LIN {X 0,Y 226.727,Z 813.985,A -85,B 0,C 180,E1 10943.796,E2 10943.796} C_VEL
LIN {X 0,Y 213.913,Z 842.664,A -85,B 0,C 180,E1 10939.312,E2 10939.312} C_VEL
LIN {X 0,Y 200.082,Z 866.438,A -85,B 0,C 180,E1 10933.575,E2 10933.575} C_VEL
LIN {X 0,Y 185.889,Z 886.486,A -85,B 0,C 180,E1 10925.902,E2 10925.902} C_VEL
LIN {X 0,Y 173.334,Z 901.965,A -85,B 0,C 180,E1 10915.797,E2 10915.797} C_VEL
LIN {X 0,Y 166.126,Z 910.389,A -85,B 0,C 180,E1 10905.806,E2 10905.806} C_VEL
LIN {X 0,Y 162.746,Z 914.405,A -85,B 0,C 180,E1 10895.312,E2 10895.312} C_VEL
LIN {X 0,Y 162.741,Z 914.431,A -85,B 0,C 180,E1 10884.671,E2 10884.671} C_VEL
LIN {X 0,Y 167.118,Z 909.261,A -85,B 0,C 180,E1 10872.286,E2 10872.286} C_VEL
LIN {X 0,Y 175.74,Z 899.256,A -85,B 0,C 180,E1 10861.809,E2 10861.809} C_VEL
LIN {X 0,Y 188.32,Z 883.429,A -85,B 0,C 180,E1 10852.545,E2 10852.545} C_VEL
LIN {X 0,Y 202.037,Z 863.615,A -85,B 0,C 180,E1 10845.474,E2 10845.474} C_VEL
LIN {X 0,Y 213.679,Z 843.483,A -85,B 0,C 180,E1 10840.733,E2 10840.733} C_VEL
LIN {X 0,Y 213.822,Z 841.755,A -85,B 0,C 180,E1 10840.089,E2 10840.089} C_VEL
LIN {X 0,Y 191.201,Z 854.023,A -85,B 0,C 180,E1 10834.887,E2 10834.887} C_VEL
LIN {X 0,Y 172.015,Z 863.269,A -85,B 0,C 180,E1 10827.408,E2 10827.408} C_VEL
LIN {X 0,Y 171.055,Z 864.24,A -85,B 0,C 180,E1 10826.511,E2 10826.511} C_VEL
LIN {X 0,Y 165.391,Z 887.788,A -85,B 0,C 180,E1 10817.921,E2 10817.921} C_VEL
LIN {X 0,Y 162.551,Z 906.246,A -85,B 0,C 180,E1 10807.992,E2 10807.992} C_VEL
LIN {X 0,Y 163.37,Z 919.553,A -85,B 0,C 180,E1 10797.341,E2 10797.341} C_VEL
LIN {X 0,Y 168.358,Z 927.831,A -85,B 0,C 180,E1 10787.041,E2 10787.041} C_VEL
LIN {X 0,Y 181.245,Z 932.296,A -85,B 0,C 180,E1 10775.39,E2 10775.39} C_VEL
LIN {X 0,Y 203.927,Z 931.055,A -85,B 0,C 180,E1 10764.501,E2 10764.501} C_VEL
LIN {X 0,Y 173.284,Z 950.433,A -85,B 0,C 180,E1 10749.162,E2 10749.162} C_VEL
LIN {X 0,Y 161.166,Z 962.439,A -85,B 0,C 180,E1 10732.005,E2 10732.005} C_VEL
LIN {X 0,Y 159.958,Z 966.188,A -85,B 0,C 180,E1 10720.884,E2 10720.884} C_VEL
LIN {X 0,Y 161.306,Z 966.713,A -85,B 0,C 180,E1 10710.008,E2 10710.008} C_VEL
LIN {X 0,Y 160.431,Z 963.91,A -85,B 0,C 180,E1 10699.165,E2 10699.165} C_VEL
LIN {X 0,Y 161.685,Z 956.022,A -85,B 0,C 180,E1 10688.087,E2 10688.087} C_VEL
LIN {X 0,Y 167.216,Z 942.935,A -85,B 0,C 180,E1 10677.225,E2 10677.225} C_VEL
LIN {X 0,Y 177.544,Z 923.702,A -85,B 0,C 180,E1 10667.168,E2 10667.168} C_VEL
LIN {X 0,Y 187.92,Z 904.945,A -85,B 0,C 180,E1 10660.657,E2 10660.657} C_VEL
LIN {X 0,Y 191.12,Z 893.404,A -85,B 0,C 180,E1 10656.782,E2 10656.782} C_VEL
LIN {X 0,Y 194.609,Z 881.1,A -85,B 0,C 180,E1 10653.221,E2 10653.221} C_VEL
LIN {X 0,Y 208.193,Z 850.796,A -85,B 0,C 180,E1 10648.474,E2 10648.474} C_VEL
LIN {X 0,Y 214.588,Z 832.369,A -85,B 0,C 180,E1 10646.423,E2 10646.423} C_VEL
LIN {X 0,Y 212.245,Z 794.393,A -85,B 0,C 180,E1 10636.132,E2 10636.132} C_VEL
LIN {X 0,Y 211.18,Z 759.787,A -85,B 0,C 180,E1 10626.677,E2 10626.677} C_VEL
LIN {X 0,Y 209.986,Z 755.134,A -85,B 0,C 180,E1 10621.038,E2 10621.038} C_VEL
LIN {X 0,Y 210.012,Z 756.128,A -85,B 0,C 180,E1 10615.631,E2 10615.631} C_VEL
LIN {X 0,Y 212.29,Z 763.26,A -85,B 0,C 180,E1 10607.698,E2 10607.698} C_VEL
LIN {X 0,Y 216.099,Z 774.144,A -85,B 0,C 180,E1 10600.64,E2 10600.64} C_VEL
LIN {X 0,Y 220.106,Z 790.379,A -85,B 0,C 180,E1 10593.547,E2 10593.547} C_VEL
LIN {X 0,Y 221.781,Z 807.929,A -85,B 0,C 180,E1 10587.791,E2 10587.791} C_VEL
LIN {X 0,Y 221.074,Z 818.297,A -85,B 0,C 180,E1 10584.988,E2 10584.988} C_VEL
LIN {X 0,Y 207.742,Z 846.1,A -85,B 0,C 180,E1 10580.508,E2 10580.508} C_VEL
LIN {X 0,Y 193.315,Z 869.391,A -85,B 0,C 180,E1 10574.624,E2 10574.624} C_VEL
LIN {X 0,Y 178.912,Z 888.584,A -85,B 0,C 180,E1 10566.924,E2 10566.924} C_VEL
LIN {X 0,Y 166.33,Z 903.215,A -85,B 0,C 180,E1 10556.969,E2 10556.969} C_VEL
LIN {X 0,Y 158.629,Z 911.638,A -85,B 0,C 180,E1 10546.574,E2 10546.574} C_VEL
LIN {X 0,Y 154.985,Z 915.652,A -85,B 0,C 180,E1 10535.579,E2 10535.579} C_VEL
LIN {X 0,Y 154.979,Z 915.678,A -85,B 0,C 180,E1 10524.404,E2 10524.404} C_VEL
LIN {X 0,Y 158.624,Z 911.712,A -85,B 0,C 180,E1 10513.408,E2 10513.408} C_VEL
LIN {X 0,Y 167.577,Z 901.928,A -85,B 0,C 180,E1 10501.776,E2 10501.776} C_VEL
LIN {X 0,Y 180.674,Z 886.595,A -85,B 0,C 180,E1 10491.966,E2 10491.966} C_VEL
LIN {X 0,Y 195.534,Z 866.419,A -85,B 0,C 180,E1 10484.319,E2 10484.319} C_VEL
LIN {X 0,Y 204.326,Z 852.412,A -85,B 0,C 180,E1 10480.722,E2 10480.722} C_VEL
LIN {X 0,Y 203.321,Z 851.933,A -85,B 0,C 180,E1 10480.046,E2 10480.046} C_VEL
LIN {X 0,Y 175.969,Z 865.016,A -85,B 0,C 180,E1 10472.393,E2 10472.393} C_VEL
LIN {X 0,Y 161.557,Z 871.91,A -85,B 0,C 180,E1 10464.839,E2 10464.839} C_VEL
LIN {X 0,Y 156.121,Z 895.313,A -85,B 0,C 180,E1 10454.816,E2 10454.816} C_VEL
LIN {X 0,Y 154.496,Z 912.023,A -85,B 0,C 180,E1 10444.188,E2 10444.188} C_VEL
LIN {X 0,Y 157.443,Z 925.022,A -85,B 0,C 180,E1 10431.723,E2 10431.723} C_VEL
LIN {X 0,Y 167.963,Z 932.703,A -85,B 0,C 180,E1 10418.928,E2 10418.928} C_VEL
LIN {X 0,Y 181.887,Z 934.6,A -85,B 0,C 180,E1 10410.137,E2 10410.137} C_VEL
LIN {X 0,Y 193.717,Z 934.19,A -85,B 0,C 180,E1 10404.961,E2 10404.961} C_VEL
LIN {X 0,Y 180.096,Z 941.694,A -85,B 0,C 180,E1 10398.961,E2 10398.961} C_VEL
LIN {X 0,Y 156.809,Z 957.546,A -85,B 0,C 180,E1 10379.977,E2 10379.977} C_VEL
LIN {X 0,Y 152.404,Z 963.144,A -85,B 0,C 180,E1 10367.29,E2 10367.29} C_VEL
LIN {X 0,Y 152.716,Z 964.845,A -85,B 0,C 180,E1 10355.68,E2 10355.68} C_VEL
LIN {X 0,Y 153.484,Z 965.461,A -85,B 0,C 180,E1 10350.009,E2 10350.009} C_VEL
LIN {X 0,Y 152.596,Z 963.789,A -85,B 0,C 180,E1 10341.501,E2 10341.501} C_VEL
LIN {X 0,Y 153.161,Z 957.796,A -85,B 0,C 180,E1 10330.686,E2 10330.686} C_VEL
LIN {X 0,Y 158.676,Z 944.628,A -85,B 0,C 180,E1 10317.784,E2 10317.784} C_VEL
LIN {X 0,Y 169.876,Z 925.215,A -85,B 0,C 180,E1 10306.502,E2 10306.502} C_VEL
LIN {X 0,Y 183.892,Z 901.354,A -85,B 0,C 180,E1 10298.019,E2 10298.019} C_VEL
LIN {X 0,Y 194.609,Z 881.1,A -85,B 0,C 180,E1 10293.221,E2 10293.221} C_VEL
LIN {X 0,Y 198.343,Z 868.128,A -85,B 0,C 180,E1 10289.936,E2 10289.936} C_VEL
LIN {X 0,Y 201.523,Z 856.291,A -85,B 0,C 180,E1 10287.312,E2 10287.312} C_VEL
LIN {X 0,Y 202.307,Z 854.439,A -85,B 0,C 180,E1 10287.059,E2 10287.059} C_VEL
LIN {X 0,Y 209.588,Z 835.114,A -85,B 0,C 180,E1 10284.745,E2 10284.745} C_VEL
LIN {X 0,Y 209.065,Z 796.132,A -85,B 0,C 180,E1 10273.869,E2 10273.869} C_VEL
LIN {X 0,Y 209.527,Z 766.811,A -85,B 0,C 180,E1 10265.433,E2 10265.433} C_VEL
LIN {X 0,Y 208.848,Z 762.923,A -85,B 0,C 180,E1 10261.044,E2 10261.044} C_VEL
LIN {X 0,Y 208.74,Z 763.849,A -85,B 0,C 180,E1 10255.994,E2 10255.994} C_VEL
LIN {X 0,Y 210.355,Z 770.807,A -85,B 0,C 180,E1 10248.108,E2 10248.108} C_VEL
LIN {X 0,Y 213.703,Z 782.943,A -85,B 0,C 180,E1 10240.319,E2 10240.319} C_VEL
LIN {X 0,Y 216.52,Z 799.927,A -85,B 0,C 180,E1 10233.076,E2 10233.076} C_VEL
LIN {X 0,Y 216.689,Z 817.671,A -85,B 0,C 180,E1 10227.318,E2 10227.318} C_VEL
LIN {X 0,Y 215.236,Z 822.861,A -85,B 0,C 180,E1 10226.235,E2 10226.235} C_VEL
LIN {X 0,Y 201.672,Z 849.417,A -85,B 0,C 180,E1 10221.775,E2 10221.775} C_VEL
LIN {X 0,Y 185.68,Z 873.66,A -85,B 0,C 180,E1 10215.318,E2 10215.318} C_VEL
LIN {X 0,Y 169.985,Z 892.966,A -85,B 0,C 180,E1 10206.746,E2 10206.746} C_VEL
LIN {X 0,Y 158.14,Z 905.758,A -85,B 0,C 180,E1 10196.945,E2 10196.945} C_VEL
LIN {X 0,Y 149.8,Z 914.308,A -85,B 0,C 180,E1 10184.578,E2 10184.578} C_VEL
LIN {X 0,Y 146.893,Z 917.424,A -85,B 0,C 180,E1 10169.991,E2 10169.991} C_VEL
LIN {X 0,Y 149.79,Z 914.373,A -85,B 0,C 180,E1 10155.403,E2 10155.403} C_VEL
LIN {X 0,Y 158.099,Z 905.884,A -85,B 0,C 180,E1 10143.029,E2 10143.029} C_VEL
LIN {X 0,Y 170.757,Z 892.19,A -85,B 0,C 180,E1 10132.662,E2 10132.662} C_VEL
LIN {X 0,Y 185.618,Z 873.941,A -85,B 0,C 180,E1 10124.643,E2 10124.643} C_VEL
LIN {X 0,Y 194.654,Z 861.037,A -85,B 0,C 180,E1 10120.801,E2 10120.801} C_VEL
LIN {X 0,Y 194.758,Z 860.103,A -85,B 0,C 180,E1 10120.335,E2 10120.335} C_VEL
LIN {X 0,Y 166.102,Z 872.724,A -85,B 0,C 180,E1 10111.475,E2 10111.475} C_VEL
LIN {X 0,Y 152.112,Z 878.872,A -85,B 0,C 180,E1 10102.977,E2 10102.977} C_VEL
LIN {X 0,Y 147.54,Z 900.094,A -85,B 0,C 180,E1 10092.559,E2 10092.559} C_VEL
LIN {X 0,Y 146.839,Z 915.669,A -85,B 0,C 180,E1 10081.459,E2 10081.459} C_VEL
LIN {X 0,Y 151.324,Z 927.878,A -85,B 0,C 180,E1 10068.484,E2 10068.484} C_VEL
LIN {X 0,Y 160.744,Z 934.107,A -85,B 0,C 180,E1 10057.934,E2 10057.934} C_VEL
LIN {X 0,Y 175.327,Z 936.65,A -85,B 0,C 180,E1 10048.899,E2 10048.899} C_VEL
LIN {X 0,Y 184.424,Z 936.772,A -85,B 0,C 180,E1 10044.924,E2 10044.924} C_VEL
LIN {X 0,Y 153.363,Z 953.588,A -85,B 0,C 180,E1 10026.196,E2 10026.196} C_VEL
LIN {X 0,Y 144.74,Z 961.456,A -85,B 0,C 180,E1 10008.237,E2 10008.237} C_VEL
LIN {X 0,Y 144.879,Z 963.376,A -85,B 0,C 180,E1 9995.988,E2 9995.988} C_VEL
LIN {X 0,Y 145.641,Z 964.206,A -85,B 0,C 180,E1 9990.009,E2 9990.009} C_VEL
LIN {X 0,Y 144.741,Z 962.518,A -85,B 0,C 180,E1 9981.036,E2 9981.036} C_VEL
LIN {X 0,Y 145.65,Z 955.918,A -85,B 0,C 180,E1 9968.842,E2 9968.842} C_VEL
LIN {X 0,Y 151.824,Z 943.101,A -85,B 0,C 180,E1 9955.962,E2 9955.962} C_VEL
LIN {X 0,Y 163.881,Z 923.872,A -85,B 0,C 180,E1 9944.479,E2 9944.479} C_VEL
LIN {X 0,Y 179.118,Z 899.607,A -85,B 0,C 180,E1 9935.789,E2 9935.789} C_VEL
LIN {X 0,Y 194.276,Z 871.816,A -85,B 0,C 180,E1 9929.669,E2 9929.669} C_VEL
LIN {X 0,Y 202.307,Z 854.439,A -85,B 0,C 180,E1 9927.059,E2 9927.059} C_VEL
LIN {X 0,Y 205,Z 843.954,A -85,B 0,C 180,E1 9924.987,E2 9924.987} C_VEL
LIN {X 0,Y 204.883,Z 828.509,A -85,B 0,C 180,E1 9920.286,E2 9920.286} C_VEL
LIN {X 0,Y 206.718,Z 788.673,A -85,B 0,C 180,E1 9908.8,E2 9908.8} C_VEL
LIN {X 0,Y 207.774,Z 773.916,A -85,B 0,C 180,E1 9904.435,E2 9904.435} C_VEL
LIN {X 0,Y 207.328,Z 770.591,A -85,B 0,C 180,E1 9900.009,E2 9900.009} C_VEL
LIN {X 0,Y 207.147,Z 771.755,A -85,B 0,C 180,E1 9896.094,E2 9896.094} C_VEL
LIN {X 0,Y 208.271,Z 778.584,A -85,B 0,C 180,E1 9888.253,E2 9888.253} C_VEL
LIN {X 0,Y 210.52,Z 789.744,A -85,B 0,C 180,E1 9881.001,E2 9881.001} C_VEL
LIN {X 0,Y 212.335,Z 806.553,A -85,B 0,C 180,E1 9873.642,E2 9873.642} C_VEL
LIN {X 0,Y 211.603,Z 822.257,A -85,B 0,C 180,E1 9868.367,E2 9868.367} C_VEL
LIN {X 0,Y 197.579,Z 849.652,A -85,B 0,C 180,E1 9863.768,E2 9863.768} C_VEL
LIN {X 0,Y 181.409,Z 873.398,A -85,B 0,C 180,E1 9857.574,E2 9857.574} C_VEL
LIN {X 0,Y 165.74,Z 892.092,A -85,B 0,C 180,E1 9849.585,E2 9849.585} C_VEL
LIN {X 0,Y 152.575,Z 905.713,A -85,B 0,C 180,E1 9839.629,E2 9839.629} C_VEL
LIN {X 0,Y 143.735,Z 914.135,A -85,B 0,C 180,E1 9828.349,E2 9828.349} C_VEL
LIN {X 0,Y 139.494,Z 918.143,A -85,B 0,C 180,E1 9816.201,E2 9816.201} C_VEL
LIN {X 0,Y 139.489,Z 918.168,A -85,B 0,C 180,E1 9803.78,E2 9803.78} C_VEL
LIN {X 0,Y 144.98,Z 913,A -85,B 0,C 180,E1 9789.461,E2 9789.461} C_VEL
LIN {X 0,Y 155.452,Z 903,A -85,B 0,C 180,E1 9777.719,E2 9777.719} C_VEL
LIN {X 0,Y 170.602,Z 886.824,A -85,B 0,C 180,E1 9767.576,E2 9767.576} C_VEL
LIN {X 0,Y 185.665,Z 867.852,A -85,B 0,C 180,E1 9760.539,E2 9760.539} C_VEL
LIN {X 0,Y 158.547,Z 878.967,A -85,B 0,C 180,E1 9751.551,E2 9751.551} C_VEL
LIN {X 0,Y 142.622,Z 886.104,A -85,B 0,C 180,E1 9740.5,E2 9740.5} C_VEL
LIN {X 0,Y 138.954,Z 906.759,A -85,B 0,C 180,E1 9728.573,E2 9728.573} C_VEL
LIN {X 0,Y 140.15,Z 922.158,A -85,B 0,C 180,E1 9715.355,E2 9715.355} C_VEL
LIN {X 0,Y 147.832,Z 932.466,A -85,B 0,C 180,E1 9702.156,E2 9702.156} C_VEL
LIN {X 0,Y 160.559,Z 937.417,A -85,B 0,C 180,E1 9691.96,E2 9691.96} C_VEL
LIN {X 0,Y 173.678,Z 938.921,A -85,B 0,C 180,E1 9685.426,E2 9685.426} C_VEL
LIN {X 0,Y 169.786,Z 940.993,A -85,B 0,C 180,E1 9683.136,E2 9683.136} C_VEL
LIN {X 0,Y 142.018,Z 955.389,A -85,B 0,C 180,E1 9662.104,E2 9662.104} C_VEL
LIN {X 0,Y 137.107,Z 959.712,A -85,B 0,C 180,E1 9649.291,E2 9649.291} C_VEL
LIN {X 0,Y 137.004,Z 962.11,A -85,B 0,C 180,E1 9636.334,E2 9636.334} C_VEL
LIN {X 0,Y 137.817,Z 962.955,A -85,B 0,C 180,E1 9630.01,E2 9630.01} C_VEL
LIN {X 0,Y 136.997,Z 961.861,A -85,B 0,C 180,E1 9622.521,E2 9622.521} C_VEL
LIN {X 0,Y 137.676,Z 955.704,A -85,B 0,C 180,E1 9609.191,E2 9609.191} C_VEL
LIN {X 0,Y 144.382,Z 942.776,A -85,B 0,C 180,E1 9594.921,E2 9594.921} C_VEL
LIN {X 0,Y 156.779,Z 924.445,A -85,B 0,C 180,E1 9583.255,E2 9583.255} C_VEL
LIN {X 0,Y 172.897,Z 900.6,A -85,B 0,C 180,E1 9574.244,E2 9574.244} C_VEL
LIN {X 0,Y 188.983,Z 873.115,A -85,B 0,C 180,E1 9567.963,E2 9567.963} C_VEL
LIN {X 0,Y 203.009,Z 843.146,A -85,B 0,C 180,E1 9563.79,E2 9563.79} C_VEL
LIN {X 0,Y 204.671,Z 838.218,A -85,B 0,C 180,E1 9563.142,E2 9563.142} C_VEL
LIN {X 0,Y 204.883,Z 828.509,A -85,B 0,C 180,E1 9560.286,E2 9560.286} C_VEL
LIN {X 0,Y 203.076,Z 823.273,A -85,B 0,C 180,E1 9557.349,E2 9557.349} C_VEL
LIN {X 0,Y 201.613,Z 818.034,A -85,B 0,C 180,E1 9554.362,E2 9554.362} C_VEL
LIN {X 0,Y 205.866,Z 781.149,A -85,B 0,C 180,E1 9543.686,E2 9543.686} C_VEL
LIN {X 0,Y 205.641,Z 778.298,A -85,B 0,C 180,E1 9540.009,E2 9540.009} C_VEL
LIN {X 0,Y 205.253,Z 779.601,A -85,B 0,C 180,E1 9536.189,E2 9536.189} C_VEL
LIN {X 0,Y 205.742,Z 785.492,A -85,B 0,C 180,E1 9529.094,E2 9529.094} C_VEL
LIN {X 0,Y 207.157,Z 796.128,A -85,B 0,C 180,E1 9521.869,E2 9521.869} C_VEL
LIN {X 0,Y 207.953,Z 811.662,A -85,B 0,C 180,E1 9514.779,E2 9514.779} C_VEL
LIN {X 0,Y 206.328,Z 826.737,A -85,B 0,C 180,E1 9509.637,E2 9509.637} C_VEL
LIN {X 0,Y 191.129,Z 853.898,A -85,B 0,C 180,E1 9504.99,E2 9504.99} C_VEL
LIN {X 0,Y 173.904,Z 877.537,A -85,B 0,C 180,E1 9498.445,E2 9498.445} C_VEL
LIN {X 0,Y 157.549,Z 895.682,A -85,B 0,C 180,E1 9490.008,E2 9490.008} C_VEL
LIN {X 0,Y 143.007,Z 909.498,A -85,B 0,C 180,E1 9478.34,E2 9478.34} C_VEL
LIN {X 0,Y 134.747,Z 916.806,A -85,B 0,C 180,E1 9466.249,E2 9466.249} C_VEL
LIN {X 0,Y 131.314,Z 919.916,A -85,B 0,C 180,E1 9449.99,E2 9449.99} C_VEL
LIN {X 0,Y 134.738,Z 916.868,A -85,B 0,C 180,E1 9433.73,E2 9433.73} C_VEL
LIN {X 0,Y 144.352,Z 908.378,A -85,B 0,C 180,E1 9420.216,E2 9420.216} C_VEL
LIN {X 0,Y 158.38,Z 894.939,A -85,B 0,C 180,E1 9409.393,E2 9409.393} C_VEL
LIN {X 0,Y 174.517,Z 876.994,A -85,B 0,C 180,E1 9401.21,E2 9401.21} C_VEL
LIN {X 0,Y 174.771,Z 875.76,A -85,B 0,C 180,E1 9400.339,E2 9400.339} C_VEL
LIN {X 0,Y 148.7,Z 885.676,A -85,B 0,C 180,E1 9390.473,E2 9390.473} C_VEL
LIN {X 0,Y 133.291,Z 892.73,A -85,B 0,C 180,E1 9377.697,E2 9377.697} C_VEL
LIN {X 0,Y 130.838,Z 911.752,A -85,B 0,C 180,E1 9364.947,E2 9364.947} C_VEL
LIN {X 0,Y 133.419,Z 925.288,A -85,B 0,C 180,E1 9351.859,E2 9351.859} C_VEL
LIN {X 0,Y 143.266,Z 935.045,A -85,B 0,C 180,E1 9338.355,E2 9338.355} C_VEL
LIN {X 0,Y 163.74,Z 940.562,A -85,B 0,C 180,E1 9325.494,E2 9325.494} C_VEL
LIN {X 0,Y 155.519,Z 944.277,A -85,B 0,C 180,E1 9320.935,E2 9320.935} C_VEL
LIN {X 0,Y 132.848,Z 955.272,A -85,B 0,C 180,E1 9300.13,E2 9300.13} C_VEL
LIN {X 0,Y 128.818,Z 959.953,A -85,B 0,C 180,E1 9280.131,E2 9280.131} C_VEL
LIN {X 0,Y 129.967,Z 961.7,A -85,B 0,C 180,E1 9270.01,E2 9270.01} C_VEL
LIN {X 0,Y 128.969,Z 959.951,A -85,B 0,C 180,E1 9259.902,E2 9259.902} C_VEL
LIN {X 0,Y 130.657,Z 952.957,A -85,B 0,C 180,E1 9245.731,E2 9245.731} C_VEL
LIN {X 0,Y 138.937,Z 939.53,A -85,B 0,C 180,E1 9231.364,E2 9231.364} C_VEL
LIN {X 0,Y 153.53,Z 920.01,A -85,B 0,C 180,E1 9219.466,E2 9219.466} C_VEL
LIN {X 0,Y 170.317,Z 896.326,A -85,B 0,C 180,E1 9211.041,E2 9211.041} C_VEL
LIN {X 0,Y 187.31,Z 867.911,A -85,B 0,C 180,E1 9205.027,E2 9205.027} C_VEL
LIN {X 0,Y 199.905,Z 840.965,A -85,B 0,C 180,E1 9201.358,E2 9201.358} C_VEL
LIN {X 0,Y 201.613,Z 818.034,A -85,B 0,C 180,E1 9194.362,E2 9194.362} C_VEL
LIN {X 0,Y 201.258,Z 808.666,A -85,B 0,C 180,E1 9190.141,E2 9190.141} C_VEL
LIN {X 0,Y 201.608,Z 799.366,A -85,B 0,C 180,E1 9185.888,E2 9185.888} C_VEL
LIN {X 0,Y 203.655,Z 787.68,A -85,B 0,C 180,E1 9182.132,E2 9182.132} C_VEL
LIN {X 0,Y 203.685,Z 785.928,A -85,B 0,C 180,E1 9180.009,E2 9180.009} C_VEL
LIN {X 0,Y 203.092,Z 787.336,A -85,B 0,C 180,E1 9176.282,E2 9176.282} C_VEL
LIN {X 0,Y 203.156,Z 793.391,A -85,B 0,C 180,E1 9168.953,E2 9168.953} C_VEL
LIN {X 0,Y 203.75,Z 804.239,A -85,B 0,C 180,E1 9161.793,E2 9161.793} C_VEL
LIN {X 0,Y 203.384,Z 819.154,A -85,B 0,C 180,E1 9154.991,E2 9154.991} C_VEL
LIN {X 0,Y 201.549,Z 829.956,A -85,B 0,C 180,E1 9151.27,E2 9151.27} C_VEL
LIN {X 0,Y 185.409,Z 857.148,A -85,B 0,C 180,E1 9146.527,E2 9146.527} C_VEL
LIN {X 0,Y 167.613,Z 880.165,A -85,B 0,C 180,E1 9139.92,E2 9139.92} C_VEL
LIN {X 0,Y 150.167,Z 898.312,A -85,B 0,C 180,E1 9131.019,E2 9131.019} C_VEL
LIN {X 0,Y 136.188,Z 910.746,A -85,B 0,C 180,E1 9119.899,E2 9119.899} C_VEL
LIN {X 0,Y 127.271,Z 918.054,A -85,B 0,C 180,E1 9107.232,E2 9107.232} C_VEL
LIN {X 0,Y 123.528,Z 921.161,A -85,B 0,C 180,E1 9089.989,E2 9089.989} C_VEL
LIN {X 0,Y 127.265,Z 918.116,A -85,B 0,C 180,E1 9072.745,E2 9072.745} C_VEL
LIN {X 0,Y 137.633,Z 909.623,A -85,B 0,C 180,E1 9058.602,E2 9058.602} C_VEL
LIN {X 0,Y 152.542,Z 896.182,A -85,B 0,C 180,E1 9047.486,E2 9047.486} C_VEL
LIN {X 0,Y 164.59,Z 883.784,A -85,B 0,C 180,E1 9041.331,E2 9041.331} C_VEL
LIN {X 0,Y 165.061,Z 882.615,A -85,B 0,C 180,E1 9040.474,E2 9040.474} C_VEL
LIN {X 0,Y 138.948,Z 891.913,A -85,B 0,C 180,E1 9029.237,E2 9029.237} C_VEL
LIN {X 0,Y 124.109,Z 899.442,A -85,B 0,C 180,E1 9014.057,E2 9014.057} C_VEL
LIN {X 0,Y 123.34,Z 917.32,A -85,B 0,C 180,E1 8999.984,E2 8999.984} C_VEL
LIN {X 0,Y 129.304,Z 930.762,A -85,B 0,C 180,E1 8984.763,E2 8984.763} C_VEL
LIN {X 0,Y 143.04,Z 939.043,A -85,B 0,C 180,E1 8971.646,E2 8971.646} C_VEL
LIN {X 0,Y 153.376,Z 941.636,A -85,B 0,C 180,E1 8965.792,E2 8965.792} C_VEL
LIN {X 0,Y 148.843,Z 943.879,A -85,B 0,C 180,E1 8962.521,E2 8962.521} C_VEL
LIN {X 0,Y 124.384,Z 954.338,A -85,B 0,C 180,E1 8939.044,E2 8939.044} C_VEL
LIN {X 0,Y 121.138,Z 957.497,A -85,B 0,C 180,E1 8924.438,E2 8924.438} C_VEL
LIN {X 0,Y 122.131,Z 960.447,A -85,B 0,C 180,E1 8910.011,E2 8910.011} C_VEL
LIN {X 0,Y 121.11,Z 958.673,A -85,B 0,C 180,E1 8899.239,E2 8899.239} C_VEL
LIN {X 0,Y 123.056,Z 951.914,A -85,B 0,C 180,E1 8884.594,E2 8884.594} C_VEL
LIN {X 0,Y 132.554,Z 938.203,A -85,B 0,C 180,E1 8869.122,E2 8869.122} C_VEL
LIN {X 0,Y 147.676,Z 919.567,A -85,B 0,C 180,E1 8857.381,E2 8857.381} C_VEL
LIN {X 0,Y 165.695,Z 895.689,A -85,B 0,C 180,E1 8848.781,E2 8848.781} C_VEL
LIN {X 0,Y 183.693,Z 867.076,A -85,B 0,C 180,E1 8842.771,E2 8842.771} C_VEL
LIN {X 0,Y 195.194,Z 844.041,A -85,B 0,C 180,E1 8839.659,E2 8839.659} C_VEL
LIN {X 0,Y 200.338,Z 807.167,A -85,B 0,C 180,E1 8828.223,E2 8828.223} C_VEL
LIN {X 0,Y 201.608,Z 799.366,A -85,B 0,C 180,E1 8825.888,E2 8825.888} C_VEL
LIN {X 0,Y 202.052,Z 794.509,A -85,B 0,C 180,E1 8823.274,E2 8823.274} C_VEL
LIN {X 0,Y 201.233,Z 793.796,A -85,B 0,C 180,E1 8819.352,E2 8819.352} C_VEL
LIN {X 0,Y 200.356,Z 798.48,A -85,B 0,C 180,E1 8811.347,E2 8811.347} C_VEL
LIN {X 0,Y 200.104,Z 809.277,A -85,B 0,C 180,E1 8803.369,E2 8803.369} C_VEL
LIN {X 0,Y 199.057,Z 823.221,A -85,B 0,C 180,E1 8796.56,E2 8796.56} C_VEL
LIN {X 0,Y 197.26,Z 832.396,A -85,B 0,C 180,E1 8793.083,E2 8793.083} C_VEL
LIN {X 0,Y 181.233,Z 858.388,A -85,B 0,C 180,E1 8788.579,E2 8788.579} C_VEL
LIN {X 0,Y 162.691,Z 881.413,A -85,B 0,C 180,E1 8782.027,E2 8782.027} C_VEL
LIN {X 0,Y 144.067,Z 899.822,A -85,B 0,C 180,E1 8772.869,E2 8772.869} C_VEL
LIN {X 0,Y 129.464,Z 911.997,A -85,B 0,C 180,E1 8761.625,E2 8761.625} C_VEL
LIN {X 0,Y 119.571,Z 919.489,A -85,B 0,C 180,E1 8747.755,E2 8747.755} C_VEL
LIN {X 0,Y 115.726,Z 922.409,A -85,B 0,C 180,E1 8729.989,E2 8729.989} C_VEL
LIN {X 0,Y 119.541,Z 919.558,A -85,B 0,C 180,E1 8712.272,E2 8712.272} C_VEL
LIN {X 0,Y 131.038,Z 910.869,A -85,B 0,C 180,E1 8696.825,E2 8696.825} C_VEL
LIN {X 0,Y 146.61,Z 897.68,A -85,B 0,C 180,E1 8685.58,E2 8685.58} C_VEL
LIN {X 0,Y 154.906,Z 889.825,A -85,B 0,C 180,E1 8681.347,E2 8681.347} C_VEL
LIN {X 0,Y 154.829,Z 889.112,A -85,B 0,C 180,E1 8680.452,E2 8680.452} C_VEL
LIN {X 0,Y 125.503,Z 899.245,A -85,B 0,C 180,E1 8664.867,E2 8664.867} C_VEL
LIN {X 0,Y 115.446,Z 905.38,A -85,B 0,C 180,E1 8650.037,E2 8650.037} C_VEL
LIN {X 0,Y 116.576,Z 922.415,A -85,B 0,C 180,E1 8634.413,E2 8634.413} C_VEL
LIN {X 0,Y 127.178,Z 935.713,A -85,B 0,C 180,E1 8617.303,E2 8617.303} C_VEL
LIN {X 0,Y 143.081,Z 942.177,A -85,B 0,C 180,E1 8606.042,E2 8606.042} C_VEL
LIN {X 0,Y 143.405,Z 942.879,A -85,B 0,C 180,E1 8604.8,E2 8604.8} C_VEL
LIN {X 0,Y 117.363,Z 952.354,A -85,B 0,C 180,E1 8580.966,E2 8580.966} C_VEL
LIN {X 0,Y 113.767,Z 954.82,A -85,B 0,C 180,E1 8569.084,E2 8569.084} C_VEL
LIN {X 0,Y 113.325,Z 958.296,A -85,B 0,C 180,E1 8557.664,E2 8557.664} C_VEL
LIN {X 0,Y 114.281,Z 959.191,A -85,B 0,C 180,E1 8550.012,E2 8550.012} C_VEL
LIN {X 0,Y 113.253,Z 957.392,A -85,B 0,C 180,E1 8538.482,E2 8538.482} C_VEL
LIN {X 0,Y 115.697,Z 950.602,A -85,B 0,C 180,E1 8522.85,E2 8522.85} C_VEL
LIN {X 0,Y 126.4,Z 936.877,A -85,B 0,C 180,E1 8506.661,E2 8506.661} C_VEL
LIN {X 0,Y 142.747,Z 918.226,A -85,B 0,C 180,E1 8494.707,E2 8494.707} C_VEL
LIN {X 0,Y 161.872,Z 894.369,A -85,B 0,C 180,E1 8486.212,E2 8486.212} C_VEL
LIN {X 0,Y 180.202,Z 866.578,A -85,B 0,C 180,E1 8480.498,E2 8480.498} C_VEL
LIN {X 0,Y 190.439,Z 847.75,A -85,B 0,C 180,E1 8478.05,E2 8478.05} C_VEL
LIN {X 0,Y 197.428,Z 811.558,A -85,B 0,C 180,E1 8466.504,E2 8466.504} C_VEL
LIN {X 0,Y 201.359,Z 794.465,A -85,B 0,C 180,E1 8461.083,E2 8461.083} C_VEL
LIN {X 0,Y 201.233,Z 793.796,A -85,B 0,C 180,E1 8459.352,E2 8459.352} C_VEL
LIN {X 0,Y 199.709,Z 797.895,A -85,B 0,C 180,E1 8455.806,E2 8455.806} C_VEL
LIN {X 0,Y 197.127,Z 807.529,A -85,B 0,C 180,E1 8450.044,E2 8450.044} C_VEL
LIN {X 0,Y 196.106,Z 818.27,A -85,B 0,C 180,E1 8442.664,E2 8442.664} C_VEL
LIN {X 0,Y 193.981,Z 831.199,A -85,B 0,C 180,E1 8436.517,E2 8436.517} C_VEL
LIN {X 0,Y 192.654,Z 835.756,A -85,B 0,C 180,E1 8434.848,E2 8434.848} C_VEL
LIN {X 0,Y 175.855,Z 861.602,A -85,B 0,C 180,E1 8430.312,E2 8430.312} C_VEL
LIN {X 0,Y 156.714,Z 884.038,A -85,B 0,C 180,E1 8423.738,E2 8423.738} C_VEL
LIN {X 0,Y 138.442,Z 901.071,A -85,B 0,C 180,E1 8415.07,E2 8415.07} C_VEL
LIN {X 0,Y 122.885,Z 913.246,A -85,B 0,C 180,E1 8403.534,E2 8403.534} C_VEL
LIN {X 0,Y 113.424,Z 919.852,A -85,B 0,C 180,E1 8391.423,E2 8391.423} C_VEL
LIN {X 0,Y 108.523,Z 923.134,A -85,B 0,C 180,E1 8377.981,E2 8377.981} C_VEL
LIN {X 0,Y 108.518,Z 923.157,A -85,B 0,C 180,E1 8361.994,E2 8361.994} C_VEL
LIN {X 0,Y 114.52,Z 919.195,A -85,B 0,C 180,E1 8346.701,E2 8346.701} C_VEL
LIN {X 0,Y 128.174,Z 909.415,A -85,B 0,C 180,E1 8331.808,E2 8331.808} C_VEL
LIN {X 0,Y 144.96,Z 895.633,A -85,B 0,C 180,E1 8321.446,E2 8321.446} C_VEL
LIN {X 0,Y 145.289,Z 894.893,A -85,B 0,C 180,E1 8320.68,E2 8320.68} C_VEL
LIN {X 0,Y 113.001,Z 906.13,A -85,B 0,C 180,E1 8299.483,E2 8299.483} C_VEL
LIN {X 0,Y 107.175,Z 911.261,A -85,B 0,C 180,E1 8285.03,E2 8285.03} C_VEL
LIN {X 0,Y 110.845,Z 927.119,A -85,B 0,C 180,E1 8268.2,E2 8268.2} C_VEL
LIN {X 0,Y 125.379,Z 939.242,A -85,B 0,C 180,E1 8251.207,E2 8251.207} C_VEL
LIN {X 0,Y 133.894,Z 942.516,A -85,B 0,C 180,E1 8245.687,E2 8245.687} C_VEL
LIN {X 0,Y 112.345,Z 949.6,A -85,B 0,C 180,E1 8226.28,E2 8226.28} C_VEL
LIN {X 0,Y 107.335,Z 951.551,A -85,B 0,C 180,E1 8214.961,E2 8214.961} C_VEL
LIN {X 0,Y 105.465,Z 957.027,A -85,B 0,C 180,E1 8198.239,E2 8198.239} C_VEL
LIN {X 0,Y 106.407,Z 957.932,A -85,B 0,C 180,E1 8190.012,E2 8190.012} C_VEL
LIN {X 0,Y 105.415,Z 956.111,A -85,B 0,C 180,E1 8177.613,E2 8177.613} C_VEL
LIN {X 0,Y 108.453,Z 949.288,A -85,B 0,C 180,E1 8160.869,E2 8160.869} C_VEL
LIN {X 0,Y 120.37,Z 935.636,A -85,B 0,C 180,E1 8144.016,E2 8144.016} C_VEL
LIN {X 0,Y 138.518,Z 916.507,A -85,B 0,C 180,E1 8131.691,E2 8131.691} C_VEL
LIN {X 0,Y 158.386,Z 893.047,A -85,B 0,C 180,E1 8123.521,E2 8123.521} C_VEL
LIN {X 0,Y 177.22,Z 865.708,A -85,B 0,C 180,E1 8118.074,E2 8118.074} C_VEL
LIN {X 0,Y 185.696,Z 851.026,A -85,B 0,C 180,E1 8116.203,E2 8116.203} C_VEL
LIN {X 0,Y 193.941,Z 818.36,A -85,B 0,C 180,E1 8105.546,E2 8105.546} C_VEL
LIN {X 0,Y 198.804,Z 801.186,A -85,B 0,C 180,E1 8100.01,E2 8100.01} C_VEL
LIN {X 0,Y 197.302,Z 806.266,A -85,B 0,C 180,E1 8091.212,E2 8091.212} C_VEL
LIN {X 0,Y 197.127,Z 807.529,A -85,B 0,C 180,E1 8090.044,E2 8090.044} C_VEL
LIN {X 0,Y 195.626,Z 814.036,A -85,B 0,C 180,E1 8086.757,E2 8086.757} C_VEL
LIN {X 0,Y 191.386,Z 827.879,A -85,B 0,C 180,E1 8081.669,E2 8081.669} C_VEL
LIN {X 0,Y 188.29,Z 839.04,A -85,B 0,C 180,E1 8076.702,E2 8076.702} C_VEL
LIN {X 0,Y 170.633,Z 864.678,A -85,B 0,C 180,E1 8072.161,E2 8072.161} C_VEL
LIN {X 0,Y 150.675,Z 886.857,A -85,B 0,C 180,E1 8065.503,E2 8065.503} C_VEL
LIN {X 0,Y 131.002,Z 903.917,A -85,B 0,C 180,E1 8056.305,E2 8056.305} C_VEL
LIN {X 0,Y 114.719,Z 915.676,A -85,B 0,C 180,E1 8043.978,E2 8043.978} C_VEL
LIN {X 0,Y 103.3,Z 922.9,A -85,B 0,C 180,E1 8026.975,E2 8026.975} C_VEL
LIN {X 0,Y 100.137,Z 924.901,A -85,B 0,C 180,E1 8009.987,E2 8009.987} C_VEL
LIN {X 0,Y 105.006,Z 921.928,A -85,B 0,C 180,E1 7989.207,E2 7989.207} C_VEL
LIN {X 0,Y 118.259,Z 913.365,A -85,B 0,C 180,E1 7972.675,E2 7972.675} C_VEL
LIN {X 0,Y 134.901,Z 901.008,A -85,B 0,C 180,E1 7961.479,E2 7961.479} C_VEL
LIN {X 0,Y 133.859,Z 900.796,A -85,B 0,C 180,E1 7960.174,E2 7960.174} C_VEL
LIN {X 0,Y 102.524,Z 912.15,A -85,B 0,C 180,E1 7933.7,E2 7933.7} C_VEL
LIN {X 0,Y 99.762,Z 916.984,A -85,B 0,C 180,E1 7918.897,E2 7918.897} C_VEL
LIN {X 0,Y 107.995,Z 932.843,A -85,B 0,C 180,E1 7899.537,E2 7899.537} C_VEL
LIN {X 0,Y 123.924,Z 942.16,A -85,B 0,C 180,E1 7885.768,E2 7885.768} C_VEL
LIN {X 0,Y 121.797,Z 943.134,A -85,B 0,C 180,E1 7883.663,E2 7883.663} C_VEL
LIN {X 0,Y 99.991,Z 950.246,A -85,B 0,C 180,E1 7856.936,E2 7856.936} C_VEL
LIN {X 0,Y 97.581,Z 955.752,A -85,B 0,C 180,E1 7838.91,E2 7838.91} C_VEL
LIN {X 0,Y 98.56,Z 956.677,A -85,B 0,C 180,E1 7830.013,E2 7830.013} C_VEL
LIN {X 0,Y 97.568,Z 954.823,A -85,B 0,C 180,E1 7816.599,E2 7816.599} C_VEL
LIN {X 0,Y 101.337,Z 947.971,A -85,B 0,C 180,E1 7798.602,E2 7798.602} C_VEL
LIN {X 0,Y 114.407,Z 934.598,A -85,B 0,C 180,E1 7781.279,E2 7781.279} C_VEL
LIN {X 0,Y 132.605,Z 916.932,A -85,B 0,C 180,E1 7769.495,E2 7769.495} C_VEL
LIN {X 0,Y 153.732,Z 893.563,A -85,B 0,C 180,E1 7761.188,E2 7761.188} C_VEL
LIN {X 0,Y 174.278,Z 865.307,A -85,B 0,C 180,E1 7755.647,E2 7755.647} C_VEL
LIN {X 0,Y 182.047,Z 852.129,A -85,B 0,C 180,E1 7753.797,E2 7753.797} C_VEL
LIN {X 0,Y 193.844,Z 814.239,A -85,B 0,C 180,E1 7741.053,E2 7741.053} C_VEL
LIN {X 0,Y 195.048,Z 810.852,A -85,B 0,C 180,E1 7740.01,E2 7740.01} C_VEL
LIN {X 0,Y 195.543,Z 809.099,A -85,B 0,C 180,E1 7738.905,E2 7738.905} C_VEL
LIN {X 0,Y 193.838,Z 814.289,A -85,B 0,C 180,E1 7730.77,E2 7730.77} C_VEL
LIN {X 0,Y 192.155,Z 823.878,A -85,B 0,C 180,E1 7723.823,E2 7723.823} C_VEL
LIN {X 0,Y 191.386,Z 827.879,A -85,B 0,C 180,E1 7721.669,E2 7721.669} C_VEL
LIN {X 0,Y 188.435,Z 835.259,A -85,B 0,C 180,E1 7719.456,E2 7719.456} C_VEL
LIN {X 0,Y 175.487,Z 855.117,A -85,B 0,C 180,E1 7716.633,E2 7716.633} C_VEL
LIN {X 0,Y 155.212,Z 879.352,A -85,B 0,C 180,E1 7711.032,E2 7711.032} C_VEL
LIN {X 0,Y 134.36,Z 898.551,A -85,B 0,C 180,E1 7703.138,E2 7703.138} C_VEL
LIN {X 0,Y 114.181,Z 913.215,A -85,B 0,C 180,E1 7691.348,E2 7691.348} C_VEL
LIN {X 0,Y 100.364,Z 921.628,A -85,B 0,C 180,E1 7676.798,E2 7676.798} C_VEL
LIN {X 0,Y 93.098,Z 925.629,A -85,B 0,C 180,E1 7659.314,E2 7659.314} C_VEL
LIN {X 0,Y 93.093,Z 925.652,A -85,B 0,C 180,E1 7640.657,E2 7640.657} C_VEL
LIN {X 0,Y 100.374,Z 921.69,A -85,B 0,C 180,E1 7623.175,E2 7623.175} C_VEL
LIN {X 0,Y 116.29,Z 911.909,A -85,B 0,C 180,E1 7607.04,E2 7607.04} C_VEL
LIN {X 0,Y 124.892,Z 905.932,A -85,B 0,C 180,E1 7601.504,E2 7601.504} C_VEL
LIN {X 0,Y 123.483,Z 905.919,A -85,B 0,C 180,E1 7599.974,E2 7599.974} C_VEL
LIN {X 0,Y 93.678,Z 917.274,A -85,B 0,C 180,E1 7569.248,E2 7569.248} C_VEL
LIN {X 0,Y 93.375,Z 922.222,A -85,B 0,C 180,E1 7551.851,E2 7551.851} C_VEL
LIN {X 0,Y 105.748,Z 936.831,A -85,B 0,C 180,E1 7532.352,E2 7532.352} C_VEL
LIN {X 0,Y 113.658,Z 941.131,A -85,B 0,C 180,E1 7526.06,E2 7526.06} C_VEL
LIN {X 0,Y 112.377,Z 942.165,A -85,B 0,C 180,E1 7523.7,E2 7523.7} C_VEL
LIN {X 0,Y 94.933,Z 946.793,A -85,B 0,C 180,E1 7503.822,E2 7503.822} C_VEL
LIN {X 0,Y 89.728,Z 953.547,A -85,B 0,C 180,E1 7484.627,E2 7484.627} C_VEL
LIN {X 0,Y 90.57,Z 955.383,A -85,B 0,C 180,E1 7469.423,E2 7469.423} C_VEL
LIN {X 0,Y 89.758,Z 953.536,A -85,B 0,C 180,E1 7455.408,E2 7455.408} C_VEL
LIN {X 0,Y 94.401,Z 946.653,A -85,B 0,C 180,E1 7435.995,E2 7435.995} C_VEL
LIN {X 0,Y 108.639,Z 933.677,A -85,B 0,C 180,E1 7418.368,E2 7418.368} C_VEL
LIN {X 0,Y 129.859,Z 914.553,A -85,B 0,C 180,E1 7405.784,E2 7405.784} C_VEL
LIN {X 0,Y 151.497,Z 891.596,A -85,B 0,C 180,E1 7398.097,E2 7398.097} C_VEL
LIN {X 0,Y 172.641,Z 863.4,A -85,B 0,C 180,E1 7392.938,E2 7392.938} C_VEL
LIN {X 0,Y 177.875,Z 854.78,A -85,B 0,C 180,E1 7391.697,E2 7391.697} C_VEL
LIN {X 0,Y 191.871,Z 817.487,A -85,B 0,C 180,E1 7378.884,E2 7378.884} C_VEL
LIN {X 0,Y 191.995,Z 816.863,A -85,B 0,C 180,E1 7377.758,E2 7377.758} C_VEL
LIN {X 0,Y 190.174,Z 821.608,A -85,B 0,C 180,E1 7370.88,E2 7370.88} C_VEL
LIN {X 0,Y 187.951,Z 830.412,A -85,B 0,C 180,E1 7364.444,E2 7364.444} C_VEL
LIN {X 0,Y 184.317,Z 842.021,A -85,B 0,C 180,E1 7358.675,E2 7358.675} C_VEL
LIN {X 0,Y 175.487,Z 855.117,A -85,B 0,C 180,E1 7356.633,E2 7356.633} C_VEL
LIN {X 0,Y 164.327,Z 868.11,A -85,B 0,C 180,E1 7355.363,E2 7355.363} C_VEL
LIN {X 0,Y 152.19,Z 880,A -85,B 0,C 180,E1 7353.782,E2 7353.782} C_VEL
LIN {X 0,Y 129.829,Z 899.798,A -85,B 0,C 180,E1 7345.895,E2 7345.895} C_VEL
LIN {X 0,Y 108.437,Z 914.465,A -85,B 0,C 180,E1 7334.077,E2 7334.077} C_VEL
LIN {X 0,Y 93.461,Z 922.877,A -85,B 0,C 180,E1 7318.957,E2 7318.957} C_VEL
LIN {X 0,Y 85.428,Z 926.874,A -85,B 0,C 180,E1 7300.159,E2 7300.159} C_VEL
LIN {X 0,Y 85.424,Z 926.896,A -85,B 0,C 180,E1 7279.809,E2 7279.809} C_VEL
LIN {X 0,Y 93.47,Z 922.938,A -85,B 0,C 180,E1 7261.014,E2 7261.014} C_VEL
LIN {X 0,Y 110.169,Z 913.483,A -85,B 0,C 180,E1 7244.638,E2 7244.638} C_VEL
LIN {X 0,Y 115.237,Z 910.092,A -85,B 0,C 180,E1 7240.873,E2 7240.873} C_VEL
LIN {X 0,Y 85.541,Z 921.801,A -85,B 0,C 180,E1 7205.037,E2 7205.037} C_VEL
LIN {X 0,Y 89.054,Z 927.897,A -85,B 0,C 180,E1 7182.729,E2 7182.729} C_VEL
LIN {X 0,Y 103.031,Z 939.365,A -85,B 0,C 180,E1 7166.667,E2 7166.667} C_VEL
LIN {X 0,Y 104.105,Z 940.557,A -85,B 0,C 180,E1 7164.544,E2 7164.544} C_VEL
LIN {X 0,Y 91.357,Z 943.068,A -85,B 0,C 180,E1 7151.376,E2 7151.376} C_VEL
LIN {X 0,Y 82.691,Z 951.045,A -85,B 0,C 180,E1 7131.424,E2 7131.424} C_VEL
LIN {X 0,Y 82.787,Z 954.155,A -85,B 0,C 180,E1 7110.016,E2 7110.016} C_VEL
LIN {X 0,Y 81.982,Z 952.247,A -85,B 0,C 180,E1 7093.988,E2 7093.988} C_VEL
LIN {X 0,Y 88.994,Z 944.154,A -85,B 0,C 180,E1 7070.533,E2 7070.533} C_VEL
LIN {X 0,Y 107.13,Z 929.618,A -85,B 0,C 180,E1 7052.331,E2 7052.331} C_VEL
LIN {X 0,Y 129.47,Z 910.386,A -85,B 0,C 180,E1 7041.206,E2 7041.206} C_VEL
LIN {X 0,Y 152.606,Z 886.281,A -85,B 0,C 180,E1 7034.177,E2 7034.177} C_VEL
LIN {X 0,Y 173.252,Z 858.803,A -85,B 0,C 180,E1 7029.905,E2 7029.905} C_VEL
LIN {X 0,Y 188.48,Z 824.073,A -85,B 0,C 180,E1 7017.716,E2 7017.716} C_VEL
LIN {X 0,Y 186.087,Z 829.209,A -85,B 0,C 180,E1 7010.678,E2 7010.678} C_VEL
LIN {X 0,Y 182.84,Z 838.765,A -85,B 0,C 180,E1 7003.998,E2 7003.998} C_VEL
LIN {X 0,Y 179.805,Z 846.007,A -85,B 0,C 180,E1 7000.584,E2 7000.584} C_VEL
LIN {X 0,Y 160.83,Z 870.811,A -85,B 0,C 180,E1 6996.164,E2 6996.164} C_VEL
LIN {X 0,Y 152.19,Z 880,A -85,B 0,C 180,E1 6993.782,E2 6993.782} C_VEL
LIN {X 0,Y 139.378,Z 890.919,A -85,B 0,C 180,E1 6991.767,E2 6991.767} C_VEL
LIN {X 0,Y 127.682,Z 899.52,A -85,B 0,C 180,E1 6989.625,E2 6989.625} C_VEL
LIN {X 0,Y 126.208,Z 900.607,A -85,B 0,C 180,E1 6989.084,E2 6989.084} C_VEL
LIN {X 0,Y 102.968,Z 915.714,A -85,B 0,C 180,E1 6977.102,E2 6977.102} C_VEL
LIN {X 0,Y 86.721,Z 924.124,A -85,B 0,C 180,E1 6961.452,E2 6961.452} C_VEL
LIN {X 0,Y 77.766,Z 928.121,A -85,B 0,C 180,E1 6941.172,E2 6941.172} C_VEL
LIN {X 0,Y 77.763,Z 928.142,A -85,B 0,C 180,E1 6918.793,E2 6918.793} C_VEL
LIN {X 0,Y 86.733,Z 924.183,A -85,B 0,C 180,E1 6898.517,E2 6898.517} C_VEL
LIN {X 0,Y 102.97,Z 915.831,A -85,B 0,C 180,E1 6882.861,E2 6882.861} C_VEL
LIN {X 0,Y 104.242,Z 914.665,A -85,B 0,C 180,E1 6880.437,E2 6880.437} C_VEL
LIN {X 0,Y 86.22,Z 932.305,A -85,B 0,C 180,E1 6814.03,E2 6814.03} C_VEL
LIN {X 0,Y 94.339,Z 938.147,A -85,B 0,C 180,E1 6805.821,E2 6805.821} C_VEL
LIN {X 0,Y 93.723,Z 938.984,A -85,B 0,C 180,E1 6803.641,E2 6803.641} C_VEL
LIN {X 0,Y 87.357,Z 940.432,A -85,B 0,C 180,E1 6797.261,E2 6797.261} C_VEL
LIN {X 0,Y 75.192,Z 949.747,A -85,B 0,C 180,E1 6773.684,E2 6773.684} C_VEL
LIN {X 0,Y 73.997,Z 951.92,A -85,B 0,C 180,E1 6761.786,E2 6761.786} C_VEL
LIN {X 0,Y 74.89,Z 952.892,A -85,B 0,C 180,E1 6750.018,E2 6750.018} C_VEL
LIN {X 0,Y 74.223,Z 950.95,A -85,B 0,C 180,E1 6732.262,E2 6732.262} C_VEL
LIN {X 0,Y 82.817,Z 942.793,A -85,B 0,C 180,E1 6706.817,E2 6706.817} C_VEL
LIN {X 0,Y 102.9,Z 928.281,A -85,B 0,C 180,E1 6688.393,E2 6688.393} C_VEL
LIN {X 0,Y 126.7,Z 909.058,A -85,B 0,C 180,E1 6677.698,E2 6677.698} C_VEL
LIN {X 0,Y 150.218,Z 885.635,A -85,B 0,C 180,E1 6671.26,E2 6671.26} C_VEL
LIN {X 0,Y 169.97,Z 860.334,A -85,B 0,C 180,E1 6667.39,E2 6667.39} C_VEL
LIN {X 0,Y 184.083,Z 832.115,A -85,B 0,C 180,E1 6657.076,E2 6657.076} C_VEL
LIN {X 0,Y 183.063,Z 833.771,A -85,B 0,C 180,E1 6653.373,E2 6653.373} C_VEL
LIN {X 0,Y 179.458,Z 841.905,A -85,B 0,C 180,E1 6646.565,E2 6646.565} C_VEL
LIN {X 0,Y 176.107,Z 849.073,A -85,B 0,C 180,E1 6642.716,E2 6642.716} C_VEL
LIN {X 0,Y 156.242,Z 873.777,A -85,B 0,C 180,E1 6638.356,E2 6638.356} C_VEL
LIN {X 0,Y 132.97,Z 895.415,A -85,B 0,C 180,E1 6631.567,E2 6631.567} C_VEL
LIN {X 0,Y 126.208,Z 900.607,A -85,B 0,C 180,E1 6629.084,E2 6629.084} C_VEL
LIN {X 0,Y 119.81,Z 904.944,A -85,B 0,C 180,E1 6627.147,E2 6627.147} C_VEL
LIN {X 0,Y 100.387,Z 915.564,A -85,B 0,C 180,E1 6622.01,E2 6622.01} C_VEL
LIN {X 0,Y 98.933,Z 916.34,A -85,B 0,C 180,E1 6621.185,E2 6621.185} C_VEL
LIN {X 0,Y 80.163,Z 925.373,A -85,B 0,C 180,E1 6604.365,E2 6604.365} C_VEL
LIN {X 0,Y 70.129,Z 929.368,A -85,B 0,C 180,E1 6582.407,E2 6582.407} C_VEL
LIN {X 0,Y 70.128,Z 929.39,A -85,B 0,C 180,E1 6557.554,E2 6557.554} C_VEL
LIN {X 0,Y 80.174,Z 925.432,A -85,B 0,C 180,E1 6535.6,E2 6535.6} C_VEL
LIN {X 0,Y 93.374,Z 919.33,A -85,B 0,C 180,E1 6522.591,E2 6522.591} C_VEL
LIN {X 0,Y 94.544,Z 918.56,A -85,B 0,C 180,E1 6520.783,E2 6520.783} C_VEL
LIN {X 0,Y 84.879,Z 936.659,A -85,B 0,C 180,E1 6445.52,E2 6445.52} C_VEL
LIN {X 0,Y 82.607,Z 938.77,A -85,B 0,C 180,E1 6442.049,E2 6442.049} C_VEL
LIN {X 0,Y 67.83,Z 948.449,A -85,B 0,C 180,E1 6416.442,E2 6416.442} C_VEL
LIN {X 0,Y 66.174,Z 950.639,A -85,B 0,C 180,E1 6403.202,E2 6403.202} C_VEL
LIN {X 0,Y 66.977,Z 951.627,A -85,B 0,C 180,E1 6390.02,E2 6390.02} C_VEL
LIN {X 0,Y 66.543,Z 949.652,A -85,B 0,C 180,E1 6370.134,E2 6370.134} C_VEL
LIN {X 0,Y 76.525,Z 941.753,A -85,B 0,C 180,E1 6343.188,E2 6343.188} C_VEL
LIN {X 0,Y 99.188,Z 926.94,A -85,B 0,C 180,E1 6324.129,E2 6324.129} C_VEL
LIN {X 0,Y 124.51,Z 907.672,A -85,B 0,C 180,E1 6314.042,E2 6314.042} C_VEL
LIN {X 0,Y 148.829,Z 884.314,A -85,B 0,C 180,E1 6308.139,E2 6308.139} C_VEL
LIN {X 0,Y 166.576,Z 862.52,A -85,B 0,C 180,E1 6304.865,E2 6304.865} C_VEL
LIN {X 0,Y 179.94,Z 838.92,A -85,B 0,C 180,E1 6295.988,E2 6295.988} C_VEL
LIN {X 0,Y 176.257,Z 845.302,A -85,B 0,C 180,E1 6289.289,E2 6289.289} C_VEL
LIN {X 0,Y 173.05,Z 851.459,A -85,B 0,C 180,E1 6285.244,E2 6285.244} C_VEL
LIN {X 0,Y 151.89,Z 876.687,A -85,B 0,C 180,E1 6280.683,E2 6280.683} C_VEL
LIN {X 0,Y 127.866,Z 897.822,A -85,B 0,C 180,E1 6274.122,E2 6274.122} C_VEL
LIN {X 0,Y 104.686,Z 913.144,A -85,B 0,C 180,E1 6264.53,E2 6264.53} C_VEL
LIN {X 0,Y 98.933,Z 916.34,A -85,B 0,C 180,E1 6261.185,E2 6261.185} C_VEL
LIN {X 0,Y 85.654,Z 922.342,A -85,B 0,C 180,E1 6255.121,E2 6255.121} C_VEL
LIN {X 0,Y 73.111,Z 926.886,A -85,B 0,C 180,E1 6246.853,E2 6246.853} C_VEL
LIN {X 0,Y 62.538,Z 930.615,A -85,B 0,C 180,E1 6223.942,E2 6223.942} C_VEL
LIN {X 0,Y 62.527,Z 930.638,A -85,B 0,C 180,E1 6196.012,E2 6196.012} C_VEL
LIN {X 0,Y 73.856,Z 926.681,A -85,B 0,C 180,E1 6172.172,E2 6172.172} C_VEL
LIN {X 0,Y 83.744,Z 922.611,A -85,B 0,C 180,E1 6162.206,E2 6162.206} C_VEL
LIN {X 0,Y 83.276,Z 922.529,A -85,B 0,C 180,E1 6160.122,E2 6160.122} C_VEL
LIN {X 0,Y 75.397,Z 938.219,A -85,B 0,C 180,E1 6085.914,E2 6085.914} C_VEL
LIN {X 0,Y 71.855,Z 940.681,A -85,B 0,C 180,E1 6080.918,E2 6080.918} C_VEL
LIN {X 0,Y 59.111,Z 948.396,A -85,B 0,C 180,E1 6052.54,E2 6052.54} C_VEL
LIN {X 0,Y 59.083,Z 950.364,A -85,B 0,C 180,E1 6030.022,E2 6030.022} C_VEL
LIN {X 0,Y 58.926,Z 948.41,A -85,B 0,C 180,E1 6007.809,E2 6007.809} C_VEL
LIN {X 0,Y 71.108,Z 940.426,A -85,B 0,C 180,E1 5978.31,E2 5978.31} C_VEL
LIN {X 0,Y 96.073,Z 925.603,A -85,B 0,C 180,E1 5959.572,E2 5959.572} C_VEL
LIN {X 0,Y 122.668,Z 906.398,A -85,B 0,C 180,E1 5950.268,E2 5950.268} C_VEL
LIN {X 0,Y 148.543,Z 882.279,A -85,B 0,C 180,E1 5944.861,E2 5944.861} C_VEL
LIN {X 0,Y 162.996,Z 865.214,A -85,B 0,C 180,E1 5942.487,E2 5942.487} C_VEL
LIN {X 0,Y 175.032,Z 846.372,A -85,B 0,C 180,E1 5935.066,E2 5935.066} C_VEL
LIN {X 0,Y 170.413,Z 853.516,A -85,B 0,C 180,E1 5928.534,E2 5928.534} C_VEL
LIN {X 0,Y 168.71,Z 856.156,A -85,B 0,C 180,E1 5927.099,E2 5927.099} C_VEL
LIN {X 0,Y 146.111,Z 881.267,A -85,B 0,C 180,E1 5922.788,E2 5922.788} C_VEL
LIN {X 0,Y 121.464,Z 901.337,A -85,B 0,C 180,E1 5916.361,E2 5916.361} C_VEL
LIN {X 0,Y 96.635,Z 916.359,A -85,B 0,C 180,E1 5906.245,E2 5906.245} C_VEL
LIN {X 0,Y 78.044,Z 924.941,A -85,B 0,C 180,E1 5892.569,E2 5892.569} C_VEL
LIN {X 0,Y 73.111,Z 926.886,A -85,B 0,C 180,E1 5886.853,E2 5886.853} C_VEL
LIN {X 0,Y 67.974,Z 928.597,A -85,B 0,C 180,E1 5881.283,E2 5881.283} C_VEL
LIN {X 0,Y 54.147,Z 932.126,A -85,B 0,C 180,E1 5861.484,E2 5861.484} C_VEL
LIN {X 0,Y 53.955,Z 932.045,A -85,B 0,C 180,E1 5860.341,E2 5860.341} C_VEL
LIN {X 0,Y 54.992,Z 931.885,A -85,B 0,C 180,E1 5834.048,E2 5834.048} C_VEL
LIN {X 0,Y 67.855,Z 927.929,A -85,B 0,C 180,E1 5808.123,E2 5808.123} C_VEL
LIN {X 0,Y 72.712,Z 926.181,A -85,B 0,C 180,E1 5803,E2 5803} C_VEL
LIN {X 0,Y 73.276,Z 925.847,A -85,B 0,C 180,E1 5800.317,E2 5800.317} C_VEL
LIN {X 0,Y 66.237,Z 939.55,A -85,B 0,C 180,E1 5726.096,E2 5726.096} C_VEL
LIN {X 0,Y 52.87,Z 946.389,A -85,B 0,C 180,E1 5701.04,E2 5701.04} C_VEL
LIN {X 0,Y 51.15,Z 949.095,A -85,B 0,C 180,E1 5670.026,E2 5670.026} C_VEL
LIN {X 0,Y 52.296,Z 946.49,A -85,B 0,C 180,E1 5640.022,E2 5640.022} C_VEL
LIN {X 0,Y 69.389,Z 937.509,A -85,B 0,C 180,E1 5609.588,E2 5609.588} C_VEL
LIN {X 0,Y 96.133,Z 922.728,A -85,B 0,C 180,E1 5593.757,E2 5593.757} C_VEL
LIN {X 0,Y 125.068,Z 902.213,A -85,B 0,C 180,E1 5585.576,E2 5585.576} C_VEL
LIN {X 0,Y 150.921,Z 877.902,A -85,B 0,C 180,E1 5581.247,E2 5581.247} C_VEL
LIN {X 0,Y 159.66,Z 867.923,A -85,B 0,C 180,E1 5580.012,E2 5580.012} C_VEL
LIN {X 0,Y 169.57,Z 853.94,A -85,B 0,C 180,E1 5574.139,E2 5574.139} C_VEL
LIN {X 0,Y 165.615,Z 859.284,A -85,B 0,C 180,E1 5569.513,E2 5569.513} C_VEL
LIN {X 0,Y 142.271,Z 884.046,A -85,B 0,C 180,E1 5565.406,E2 5565.406} C_VEL
LIN {X 0,Y 116.894,Z 903.723,A -85,B 0,C 180,E1 5559.352,E2 5559.352} C_VEL
LIN {X 0,Y 91.127,Z 918.276,A -85,B 0,C 180,E1 5549.585,E2 5549.585} C_VEL
LIN {X 0,Y 67.841,Z 927.873,A -85,B 0,C 180,E1 5531.835,E2 5531.835} C_VEL
LIN {X 0,Y 54.999,Z 931.863,A -85,B 0,C 180,E1 5505.9,E2 5505.9} C_VEL
LIN {X 0,Y 53.955,Z 932.045,A -85,B 0,C 180,E1 5500.341,E2 5500.341} C_VEL
LIN {X 0,Y 50.811,Z 932.775,A -85,B 0,C 180,E1 5486.367,E2 5486.367} C_VEL
LIN {X 0,Y 50.357,Z 932.459,A -85,B 0,C 180,E1 5462.422,E2 5462.422} C_VEL
LIN {X 0,Y 50.802,Z 932.233,A -85,B 0,C 180,E1 5461.28,E2 5461.28} C_VEL
LIN {X 0,Y 62.261,Z 929.176,A -85,B 0,C 180,E1 5443.322,E2 5443.322} C_VEL
LIN {X 0,Y 63.286,Z 928.819,A -85,B 0,C 180,E1 5440.553,E2 5440.553} C_VEL
LIN {X 0,Y 56.152,Z 940.402,A -85,B 0,C 180,E1 5367.451,E2 5367.451} C_VEL
LIN {X 0,Y 55.427,Z 941.106,A -85,B 0,C 180,E1 5364.807,E2 5364.807} C_VEL
LIN {X 0,Y 43.031,Z 946.78,A -85,B 0,C 180,E1 5330.563,E2 5330.563} C_VEL
LIN {X 0,Y 43.232,Z 947.829,A -85,B 0,C 180,E1 5310.03,E2 5310.03} C_VEL
LIN {X 0,Y 45.043,Z 945.365,A -85,B 0,C 180,E1 5276.282,E2 5276.282} C_VEL
LIN {X 0,Y 65.686,Z 936.181,A -85,B 0,C 180,E1 5243.275,E2 5243.275} C_VEL
LIN {X 0,Y 92.879,Z 922.362,A -85,B 0,C 180,E1 5229.37,E2 5229.37} C_VEL
LIN {X 0,Y 122.672,Z 902.313,A -85,B 0,C 180,E1 5222.104,E2 5222.104} C_VEL
LIN {X 0,Y 150.013,Z 877.586,A -85,B 0,C 180,E1 5218.222,E2 5218.222} C_VEL
LIN {X 0,Y 157.003,Z 869.829,A -85,B 0,C 180,E1 5217.15,E2 5217.15} C_VEL
LIN {X 0,Y 163.272,Z 861.925,A -85,B 0,C 180,E1 5213.904,E2 5213.904} C_VEL
LIN {X 0,Y 162.459,Z 862.854,A -85,B 0,C 180,E1 5212.128,E2 5212.128} C_VEL
LIN {X 0,Y 138.733,Z 886.815,A -85,B 0,C 180,E1 5208.185,E2 5208.185} C_VEL
LIN {X 0,Y 112.669,Z 906.04,A -85,B 0,C 180,E1 5202.576,E2 5202.576} C_VEL
LIN {X 0,Y 84.821,Z 920.72,A -85,B 0,C 180,E1 5192.785,E2 5192.785} C_VEL
LIN {X 0,Y 62.243,Z 929.121,A -85,B 0,C 180,E1 5176.634,E2 5176.634} C_VEL
LIN {X 0,Y 46.832,Z 933.287,A -85,B 0,C 180,E1 5145.016,E2 5145.016} C_VEL
LIN {X 0,Y 47.535,Z 933.133,A -85,B 0,C 180,E1 5111.461,E2 5111.461} C_VEL
LIN {X 0,Y 50.802,Z 932.233,A -85,B 0,C 180,E1 5101.28,E2 5101.28} C_VEL
LIN {X 0,Y 52.475,Z 931.795,A -85,B 0,C 180,E1 5091.039,E2 5091.039} C_VEL
LIN {X 0,Y 50.649,Z 932.135,A -85,B 0,C 180,E1 5078.836,E2 5078.836} C_VEL
LIN {X 0,Y 48.545,Z 932.703,A -85,B 0,C 180,E1 5073.968,E2 5073.968} C_VEL
LIN {X 0,Y 45.663,Z 940.787,A -85,B 0,C 180,E1 5010.239,E2 5010.239} C_VEL
LIN {X 0,Y 45.823,Z 941.69,A -85,B 0,C 180,E1 5005.468,E2 5005.468} C_VEL
LIN {X 0,Y 35.591,Z 945.49,A -85,B 0,C 180,E1 4975.128,E2 4975.128} C_VEL
LIN {X 0,Y 35.264,Z 946.555,A -85,B 0,C 180,E1 4950.037,E2 4950.037} C_VEL
LIN {X 0,Y 37.263,Z 944.565,A -85,B 0,C 180,E1 4914.169,E2 4914.169} C_VEL
LIN {X 0,Y 59.647,Z 936.191,A -85,B 0,C 180,E1 4878.492,E2 4878.492} C_VEL
LIN {X 0,Y 90.803,Z 921.6,A -85,B 0,C 180,E1 4864.513,E2 4864.513} C_VEL
LIN {X 0,Y 120.745,Z 902.399,A -85,B 0,C 180,E1 4858.494,E2 4858.494} C_VEL
LIN {X 0,Y 148.564,Z 878.266,A -85,B 0,C 180,E1 4855.258,E2 4855.258} C_VEL
LIN {X 0,Y 154.354,Z 872.186,A -85,B 0,C 180,E1 4854.403,E2 4854.403} C_VEL
LIN {X 0,Y 151.877,Z 874.617,A -85,B 0,C 180,E1 4853.449,E2 4853.449} C_VEL
LIN {X 0,Y 125.846,Z 897.131,A -85,B 0,C 180,E1 4849.496,E2 4849.496} C_VEL
LIN {X 0,Y 98.385,Z 914.114,A -85,B 0,C 180,E1 4843.42,E2 4843.42} C_VEL
LIN {X 0,Y 68.819,Z 926.736,A -85,B 0,C 180,E1 4831.258,E2 4831.258} C_VEL
LIN {X 0,Y 47.303,Z 932.875,A -85,B 0,C 180,E1 4809.61,E2 4809.61} C_VEL
LIN {X 0,Y 37.828,Z 934.866,A -85,B 0,C 180,E1 4769.965,E2 4769.965} C_VEL
LIN {X 0,Y 51.992,Z 931.825,A -85,B 0,C 180,E1 4723.403,E2 4723.403} C_VEL
LIN {X 0,Y 52.971,Z 931.536,A -85,B 0,C 180,E1 4720.481,E2 4720.481} C_VEL
LIN {X 0,Y 48.545,Z 932.703,A -85,B 0,C 180,E1 4713.968,E2 4713.968} C_VEL
LIN {X 0,Y 37.716,Z 936.119,A -85,B 0,C 180,E1 4695.992,E2 4695.992} C_VEL
LIN {X 0,Y 32.784,Z 939.443,A -85,B 0,C 180,E1 4668.852,E2 4668.852} C_VEL
LIN {X 0,Y 35.342,Z 940.882,A -85,B 0,C 180,E1 4654.666,E2 4654.666} C_VEL
LIN {X 0,Y 36.231,Z 941.939,A -85,B 0,C 180,E1 4646.478,E2 4646.478} C_VEL
LIN {X 0,Y 27.294,Z 945.28,A -85,B 0,C 180,E1 4590.048,E2 4590.048} C_VEL
LIN {X 0,Y 31.002,Z 943.256,A -85,B 0,C 180,E1 4545.28,E2 4545.28} C_VEL
LIN {X 0,Y 57.549,Z 934.857,A -85,B 0,C 180,E1 4510.598,E2 4510.598} C_VEL
LIN {X 0,Y 90.53,Z 920.262,A -85,B 0,C 180,E1 4499.225,E2 4499.225} C_VEL
LIN {X 0,Y 121.248,Z 901.073,A -85,B 0,C 180,E1 4494.568,E2 4494.568} C_VEL
LIN {X 0,Y 127.024,Z 896.746,A -85,B 0,C 180,E1 4494.005,E2 4494.005} C_VEL
LIN {X 0,Y 122.6,Z 899.793,A -85,B 0,C 180,E1 4492.717,E2 4492.717} C_VEL
LIN {X 0,Y 92.9,Z 917.118,A -85,B 0,C 180,E1 4487.007,E2 4487.007} C_VEL
LIN {X 0,Y 65.42,Z 927.986,A -85,B 0,C 180,E1 4477.273,E2 4477.273} C_VEL
LIN {X 0,Y 41.595,Z 934.122,A -85,B 0,C 180,E1 4456.474,E2 4456.474} C_VEL
LIN {X 0,Y 30.026,Z 936.114,A -85,B 0,C 180,E1 4409.956,E2 4409.956} C_VEL
LIN {X 0,Y 41.626,Z 934.163,A -85,B 0,C 180,E1 4363.48,E2 4363.48} C_VEL
LIN {X 0,Y 42.199,Z 934.074,A -85,B 0,C 180,E1 4359.681,E2 4359.681} C_VEL
LIN {X 0,Y 32.784,Z 939.443,A -85,B 0,C 180,E1 4308.852,E2 4308.852} C_VEL
LIN {X 0,Y 30.858,Z 940.914,A -85,B 0,C 180,E1 4297.257,E2 4297.257} C_VEL
LIN {X 0,Y 23.809,Z 942.633,A -85,B 0,C 180,E1 4279.144,E2 4279.144} C_VEL
LIN {X 0,Y 20.317,Z 943.18,A -85,B 0,C 180,E1 4263.88,E2 4263.88} C_VEL
LIN {X 0,Y 19.291,Z 944.001,A -85,B 0,C 180,E1 4230.068,E2 4230.068} C_VEL
LIN {X 0,Y 26.799,Z 941.707,A -85,B 0,C 180,E1 4169.88,E2 4169.88} C_VEL
LIN {X 0,Y 56.612,Z 933.523,A -85,B 0,C 180,E1 4142.269,E2 4142.269} C_VEL
LIN {X 0,Y 91.024,Z 918.932,A -85,B 0,C 180,E1 4133.981,E2 4133.981} C_VEL
LIN {X 0,Y 96.571,Z 915.971,A -85,B 0,C 180,E1 4133.278,E2 4133.278} C_VEL
LIN {X 0,Y 73.4,Z 925.762,A -85,B 0,C 180,E1 4127.495,E2 4127.495} C_VEL
LIN {X 0,Y 42.741,Z 934.279,A -85,B 0,C 180,E1 4111.904,E2 4111.904} C_VEL
LIN {X 0,Y 22.239,Z 937.359,A -85,B 0,C 180,E1 4049.941,E2 4049.941} C_VEL
LIN {X 0,Y 30.764,Z 936.315,A -85,B 0,C 180,E1 4003.852,E2 4003.852} C_VEL
LIN {X 0,Y 31.54,Z 936.29,A -85,B 0,C 180,E1 3998.862,E2 3998.862} C_VEL
LIN {X 0,Y 26.757,Z 941.305,A -85,B 0,C 180,E1 3934.9,E2 3934.9} C_VEL
LIN {X 0,Y 26.439,Z 941.951,A -85,B 0,C 180,E1 3927.816,E2 3927.816} C_VEL
LIN {X 0,Y 20.317,Z 943.18,A -85,B 0,C 180,E1 3903.88,E2 3903.88} C_VEL
LIN {X 0,Y 15.937,Z 943.459,A -85,B 0,C 180,E1 3872.088,E2 3872.088} C_VEL
LIN {X 0,Y 22.826,Z 940.555,A -85,B 0,C 180,E1 3793.82,E2 3793.82} C_VEL
LIN {X 0,Y 56.895,Z 932.189,A -85,B 0,C 180,E1 3773.845,E2 3773.845} C_VEL
LIN {X 0,Y 64.169,Z 929.682,A -85,B 0,C 180,E1 3772.363,E2 3772.363} C_VEL
LIN {X 0,Y 32.866,Z 936.615,A -85,B 0,C 180,E1 3756.581,E2 3756.581} C_VEL
LIN {X 0,Y 14.448,Z 938.605,A -85,B 0,C 180,E1 3689.909,E2 3689.909} C_VEL
LIN {X 0,Y 20.548,Z 938.113,A -85,B 0,C 180,E1 3642.647,E2 3642.647} C_VEL
LIN {X 0,Y 16.671,Z 940.238,A -85,B 0,C 180,E1 3599.884,E2 3599.884} C_VEL
LIN {X 0,Y 17.081,Z 941.611,A -85,B 0,C 180,E1 3572.232,E2 3572.232} C_VEL
LIN {X 0,Y 11.273,Z 942.718,A -85,B 0,C 180,E1 3510.117,E2 3510.117} C_VEL
LIN {X 0,Y 22.826,Z 940.555,A -85,B 0,C 180,E1 3433.82,E2 3433.82} C_VEL
LIN {X 0,Y 21.475,Z 940.085,A -85,B 0,C 180,E1 3424.578,E2 3424.578} C_VEL
LIN {X 0,Y 14.42,Z 939.899,A -85,B 0,C 180,E1 3407.001,E2 3407.001} C_VEL
LIN {X 0,Y 6.897,Z 939.781,A -85,B 0,C 180,E1 3347.174,E2 3347.174} C_VEL
LIN {X 0,Y 9.182,Z 939.749,A -85,B 0,C 180,E1 3284.492,E2 3284.492} C_VEL
LIN {X 0,Y 10.005,Z 939.955,A -85,B 0,C 180,E1 3268.902,E2 3268.902} C_VEL
LIN {X 0,Y 8.64,Z 940.736,A -85,B 0,C 180,E1 3239.777,E2 3239.777} C_VEL
LIN {X 0,Y 3.236,Z 941.433,A -85,B 0,C 180,E1 3150.407,E2 3150.407} C_VEL
LIN {X 0,Y 28.026,Z 938.343,A -85,B 0,C 180,E1 3050.639,E2 3050.639} C_VEL
LIN {X 0,Y 6.897,Z 939.781,A -85,B 0,C 180,E1 2987.174,E2 2987.174} C_VEL
LIN {X 0,Y 6.657,Z 941.78,A -85,B 0,C 180,E1 2970.904,E2 2970.904} C_VEL
LIN {X 0,Y 6.657,Z 1015.5,A -85,B 0,C 180,E1 2970.904,E2 2970.904} C_VEL
LIN {X 0,Y 6.657,Z 1015.5,A -85,B 0,C 180,E1 2970.904,E2 2970.904}

QRS_NEXT_CUT()
PTP {E1 3056.924,E2 3056.924}
PTP {X 0,Y 607.924,A -85,B 0,C 180,E1 3056.924,E2 3056.924,E3 0,E4 0,E5 0,E6 0}
QRS_SPEED_INIT()
LIN {X 0,Y 607.924,Z 1015.5,A -85,B 0,C 180,E1 3056.924,E2 3056.924,E3 0,E4 0,E5 0,E6 0} C_VEL
LIN {X 0,Y 607.924,Z 365.092,A -85,B 0,C 180,E1 3056.924,E2 3056.924} C_VEL
LIN {X 0,Y 607.924,Z 357.014,A -85,B 0,C 180,E1 3056.924,E2 3056.924} C_VEL
LIN {X 0,Y 607.899,Z 355.014,A -85,B 0,C 180,E1 3056.736,E2 3056.736} C_VEL
LIN {X 0,Y 607.91,Z 355.014,A -85,B 0,C 180,E1 3053.578,E2 3053.578} C_VEL
LIN {X 0,Y 607.915,Z 355.015,A -85,B 0,C 180,E1 3050.438,E2 3050.438} C_VEL
LIN {X 0,Y 607.912,Z 355.015,A -85,B 0,C 180,E1 3047.247,E2 3047.247} C_VEL
LIN {X 0,Y 607.914,Z 355.014,A -85,B 0,C 180,E1 3044.057,E2 3044.057} C_VEL
LIN {X 0,Y 607.895,Z 355.015,A -85,B 0,C 180,E1 3040.894,E2 3040.894} C_VEL
LIN {X 0,Y 607.906,Z 355.012,A -85,B 0,C 180,E1 3037.772,E2 3037.772} C_VEL
LIN {X 0,Y 607.87,Z 355.015,A -85,B 0,C 180,E1 3034.68,E2 3034.68} C_VEL
LIN {X 0,Y 607.891,Z 355.012,A -85,B 0,C 180,E1 3031.511,E2 3031.511} C_VEL
LIN {X 0,Y 607.873,Z 355.013,A -85,B 0,C 180,E1 3028.572,E2 3028.572} C_VEL
LIN {X 0,Y 607.877,Z 355.012,A -85,B 0,C 180,E1 3025.311,E2 3025.311} C_VEL
LIN {X 0,Y 607.89,Z 355.011,A -85,B 0,C 180,E1 3022.275,E2 3022.275} C_VEL
LIN {X 0,Y 607.867,Z 355.015,A -85,B 0,C 180,E1 3019.106,E2 3019.106} C_VEL
LIN {X 0,Y 607.903,Z 355.012,A -85,B 0,C 180,E1 3016.045,E2 3016.045} C_VEL
LIN {X 0,Y 607.892,Z 355.015,A -85,B 0,C 180,E1 3012.917,E2 3012.917} C_VEL
LIN {X 0,Y 607.915,Z 355.013,A -85,B 0,C 180,E1 3009.777,E2 3009.777} C_VEL
LIN {X 0,Y 607.906,Z 355.015,A -85,B 0,C 180,E1 3006.541,E2 3006.541} C_VEL
LIN {X 0,Y 607.919,Z 355.014,A -85,B 0,C 180,E1 3003.321,E2 3003.321} C_VEL
LIN {X 0,Y 607.909,Z 355.129,A -85,B 0,C 180,E1 3000.088,E2 3000.088} C_VEL
LIN {X 0,Y 607.916,Z 400.904,A -85,B 0,C 180,E1 2996.997,E2 2996.997} C_VEL
LIN {X 0,Y 607.899,Z 448.599,A -85,B 0,C 180,E1 2993.865,E2 2993.865} C_VEL
LIN {X 0,Y 607.906,Z 473.153,A -85,B 0,C 180,E1 2992.285,E2 2992.285} C_VEL
LIN {X 0,Y 607.914,Z 682.432,A -85,B 0,C 180,E1 2989.667,E2 2989.667} C_VEL
LIN {X 0,Y 607.915,Z 701.405,A -85,B 0,C 180,E1 2989.251,E2 2989.251} C_VEL
LIN {X 0,Y 607.917,Z 719.664,A -85,B 0,C 180,E1 2988.672,E2 2988.672} C_VEL
LIN {X 0,Y 607.883,Z 737.661,A -85,B 0,C 180,E1 2987.913,E2 2987.913} C_VEL
LIN {X 0,Y 607.919,Z 754.368,A -85,B 0,C 180,E1 2987.023,E2 2987.023} C_VEL
LIN {X 0,Y 607.917,Z 770.201,A -85,B 0,C 180,E1 2985.991,E2 2985.991} C_VEL
LIN {X 0,Y 607.915,Z 785.11,A -85,B 0,C 180,E1 2984.818,E2 2984.818} C_VEL
LIN {X 0,Y 607.915,Z 799.021,A -85,B 0,C 180,E1 2983.506,E2 2983.506} C_VEL
LIN {X 0,Y 607.916,Z 811.823,A -85,B 0,C 180,E1 2982.057,E2 2982.057} C_VEL
LIN {X 0,Y 607.915,Z 823.066,A -85,B 0,C 180,E1 2980.519,E2 2980.519} C_VEL
LIN {X 0,Y 607.914,Z 832.765,A -85,B 0,C 180,E1 2978.894,E2 2978.894} C_VEL
LIN {X 0,Y 607.909,Z 840.488,A -85,B 0,C 180,E1 2977.276,E2 2977.276} C_VEL
LIN {X 0,Y 607.907,Z 846.767,A -85,B 0,C 180,E1 2975.569,E2 2975.569} C_VEL
LIN {X 0,Y 607.918,Z 851.275,A -85,B 0,C 180,E1 2973.866,E2 2973.866} C_VEL
LIN {X 0,Y 607.916,Z 854.234,A -85,B 0,C 180,E1 2972.073,E2 2972.073} C_VEL
LIN {X 0,Y 607.908,Z 855.429,A -85,B 0,C 180,E1 2970.282,E2 2970.282} C_VEL
LIN {X 0,Y 607.915,Z 854.879,A -85,B 0,C 180,E1 2968.492,E2 2968.492} C_VEL
LIN {X 0,Y 607.909,Z 852.579,A -85,B 0,C 180,E1 2966.7,E2 2966.7} C_VEL
LIN {X 0,Y 607.905,Z 848.715,A -85,B 0,C 180,E1 2964.999,E2 2964.999} C_VEL
LIN {X 0,Y 607.911,Z 843.133,A -85,B 0,C 180,E1 2963.294,E2 2963.294} C_VEL
LIN {X 0,Y 607.916,Z 836.139,A -85,B 0,C 180,E1 2961.678,E2 2961.678} C_VEL
LIN {X 0,Y 607.911,Z 827.279,A -85,B 0,C 180,E1 2960.055,E2 2960.055} C_VEL
LIN {X 0,Y 607.917,Z 816.973,A -85,B 0,C 180,E1 2958.521,E2 2958.521} C_VEL
LIN {X 0,Y 607.913,Z 805.239,A -85,B 0,C 180,E1 2957.074,E2 2957.074} C_VEL
LIN {X 0,Y 607.917,Z 792.055,A -85,B 0,C 180,E1 2955.717,E2 2955.717} C_VEL
LIN {X 0,Y 607.917,Z 777.294,A -85,B 0,C 180,E1 2954.449,E2 2954.449} C_VEL
LIN {X 0,Y 607.918,Z 761.431,A -85,B 0,C 180,E1 2953.321,E2 2953.321} C_VEL
LIN {X 0,Y 607.894,Z 744.425,A -85,B 0,C 180,E1 2952.334,E2 2952.334} C_VEL
LIN {X 0,Y 607.904,Z 727.427,A -85,B 0,C 180,E1 2951.541,E2 2951.541} C_VEL
LIN {X 0,Y 607.914,Z 709.536,A -85,B 0,C 180,E1 2950.895,E2 2950.895} C_VEL
LIN {X 0,Y 607.911,Z 691.218,A -85,B 0,C 180,E1 2950.413,E2 2950.413} C_VEL
LIN {X 0,Y 607.912,Z 672.235,A -85,B 0,C 180,E1 2950.095,E2 2950.095} C_VEL
LIN {X 0,Y 607.909,Z 473.031,A -85,B 0,C 180,E1 2947.621,E2 2947.621} C_VEL
LIN {X 0,Y 607.907,Z 425.103,A -85,B 0,C 180,E1 2944.512,E2 2944.512} C_VEL
LIN {X 0,Y 607.918,Z 378.396,A -85,B 0,C 180,E1 2941.405,E2 2941.405} C_VEL
LIN {X 0,Y 607.864,Z 355.016,A -85,B 0,C 180,E1 2939.806,E2 2939.806} C_VEL
LIN {X 0,Y 607.871,Z 355.01,A -85,B 0,C 180,E1 2936.506,E2 2936.506} C_VEL
LIN {X 0,Y 607.864,Z 355.013,A -85,B 0,C 180,E1 2933.573,E2 2933.573} C_VEL
LIN {X 0,Y 607.865,Z 355.01,A -85,B 0,C 180,E1 2930.219,E2 2930.219} C_VEL
LIN {X 0,Y 607.866,Z 355.013,A -85,B 0,C 180,E1 2927.329,E2 2927.329} C_VEL
LIN {X 0,Y 607.865,Z 355.01,A -85,B 0,C 180,E1 2924.043,E2 2924.043} C_VEL
LIN {X 0,Y 607.866,Z 355.013,A -85,B 0,C 180,E1 2921.118,E2 2921.118} C_VEL
LIN {X 0,Y 607.867,Z 355.01,A -85,B 0,C 180,E1 2917.846,E2 2917.846} C_VEL
LIN {X 0,Y 607.864,Z 355.014,A -85,B 0,C 180,E1 2914.919,E2 2914.919} C_VEL
LIN {X 0,Y 607.891,Z 355.221,A -85,B 0,C 180,E1 2911.869,E2 2911.869} C_VEL
LIN {X 0,Y 607.902,Z 394.047,A -85,B 0,C 180,E1 2909.026,E2 2909.026} C_VEL
LIN {X 0,Y 607.917,Z 438.431,A -85,B 0,C 180,E1 2905.885,E2 2905.885} C_VEL
LIN {X 0,Y 607.906,Z 484.105,A -85,B 0,C 180,E1 2902.738,E2 2902.738} C_VEL
LIN {X 0,Y 607.91,Z 531.711,A -85,B 0,C 180,E1 2899.534,E2 2899.534} C_VEL
LIN {X 0,Y 607.902,Z 580.177,A -85,B 0,C 180,E1 2896.335,E2 2896.335} C_VEL
LIN {X 0,Y 607.9,Z 588.718,A -85,B 0,C 180,E1 2895.793,E2 2895.793} C_VEL
LIN {X 0,Y 607.897,Z 731.168,A -85,B 0,C 180,E1 2894.065,E2 2894.065} C_VEL
LIN {X 0,Y 607.903,Z 748.009,A -85,B 0,C 180,E1 2893.677,E2 2893.677} C_VEL
LIN {X 0,Y 607.907,Z 762.769,A -85,B 0,C 180,E1 2893.169,E2 2893.169} C_VEL
LIN {X 0,Y 607.914,Z 777.332,A -85,B 0,C 180,E1 2892.491,E2 2892.491} C_VEL
LIN {X 0,Y 607.918,Z 791.757,A -85,B 0,C 180,E1 2891.624,E2 2891.624} C_VEL
LIN {X 0,Y 607.919,Z 804.432,A -85,B 0,C 180,E1 2890.663,E2 2890.663} C_VEL
LIN {X 0,Y 607.918,Z 817.049,A -85,B 0,C 180,E1 2889.467,E2 2889.467} C_VEL
LIN {X 0,Y 607.916,Z 827.44,A -85,B 0,C 180,E1 2888.227,E2 2888.227} C_VEL
LIN {X 0,Y 607.917,Z 836.325,A -85,B 0,C 180,E1 2886.896,E2 2886.896} C_VEL
LIN {X 0,Y 607.914,Z 843.658,A -85,B 0,C 180,E1 2885.474,E2 2885.474} C_VEL
LIN {X 0,Y 607.914,Z 849.35,A -85,B 0,C 180,E1 2883.961,E2 2883.961} C_VEL
LIN {X 0,Y 607.915,Z 853.151,A -85,B 0,C 180,E1 2882.451,E2 2882.451} C_VEL
LIN {X 0,Y 607.916,Z 855.103,A -85,B 0,C 180,E1 2880.943,E2 2880.943} C_VEL
LIN {X 0,Y 607.913,Z 855.358,A -85,B 0,C 180,E1 2879.341,E2 2879.341} C_VEL
LIN {X 0,Y 607.918,Z 853.773,A -85,B 0,C 180,E1 2877.832,E2 2877.832} C_VEL
LIN {X 0,Y 607.915,Z 850.464,A -85,B 0,C 180,E1 2876.323,E2 2876.323} C_VEL
LIN {X 0,Y 607.916,Z 845.662,A -85,B 0,C 180,E1 2874.905,E2 2874.905} C_VEL
LIN {X 0,Y 607.916,Z 838.962,A -85,B 0,C 180,E1 2873.484,E2 2873.484} C_VEL
LIN {X 0,Y 607.916,Z 830.84,A -85,B 0,C 180,E1 2872.154,E2 2872.154} C_VEL
LIN {X 0,Y 607.917,Z 821.285,A -85,B 0,C 180,E1 2870.916,E2 2870.916} C_VEL
LIN {X 0,Y 607.918,Z 809.262,A -85,B 0,C 180,E1 2869.673,E2 2869.673} C_VEL
LIN {X 0,Y 607.919,Z 797.082,A -85,B 0,C 180,E1 2868.665,E2 2868.665} C_VEL
LIN {X 0,Y 607.904,Z 783.268,A -85,B 0,C 180,E1 2867.75,E2 2867.75} C_VEL
LIN {X 0,Y 607.906,Z 769.424,A -85,B 0,C 180,E1 2867.026,E2 2867.026} C_VEL
LIN {X 0,Y 607.912,Z 754.006,A -85,B 0,C 180,E1 2866.421,E2 2866.421} C_VEL
LIN {X 0,Y 607.894,Z 738.217,A -85,B 0,C 180,E1 2865.984,E2 2865.984} C_VEL
LIN {X 0,Y 607.901,Z 721.471,A -85,B 0,C 180,E1 2865.708,E2 2865.708} C_VEL
LIN {X 0,Y 607.899,Z 588.32,A -85,B 0,C 180,E1 2864.106,E2 2864.106} C_VEL
LIN {X 0,Y 607.906,Z 541.01,A -85,B 0,C 180,E1 2860.995,E2 2860.995} C_VEL
LIN {X 0,Y 607.905,Z 494.449,A -85,B 0,C 180,E1 2857.874,E2 2857.874} C_VEL
LIN {X 0,Y 607.913,Z 449.156,A -85,B 0,C 180,E1 2854.771,E2 2854.771} C_VEL
LIN {X 0,Y 607.908,Z 403.572,A -85,B 0,C 180,E1 2851.566,E2 2851.566} C_VEL
LIN {X 0,Y 607.91,Z 375.546,A -85,B 0,C 180,E1 2849.525,E2 2849.525} C_VEL
LIN {X 0,Y 607.881,Z 355.015,A -85,B 0,C 180,E1 2847.513,E2 2847.513} C_VEL
LIN {X 0,Y 607.89,Z 355.014,A -85,B 0,C 180,E1 2844.507,E2 2844.507} C_VEL
LIN {X 0,Y 607.882,Z 355.014,A -85,B 0,C 180,E1 2841.316,E2 2841.316} C_VEL
LIN {X 0,Y 607.903,Z 355.239,A -85,B 0,C 180,E1 2839.124,E2 2839.124} C_VEL
LIN {X 0,Y 607.913,Z 416.266,A -85,B 0,C 180,E1 2836.046,E2 2836.046} C_VEL
LIN {X 0,Y 607.902,Z 429.394,A -85,B 0,C 180,E1 2835.2,E2 2835.2} C_VEL
LIN {X 0,Y 607.91,Z 437.617,A -85,B 0,C 180,E1 2834.481,E2 2834.481} C_VEL
LIN {X 0,Y 607.891,Z 442.025,A -85,B 0,C 180,E1 2833.911,E2 2833.911} C_VEL
LIN {X 0,Y 607.914,Z 443.592,A -85,B 0,C 180,E1 2833.504,E2 2833.504} C_VEL
LIN {X 0,Y 607.896,Z 443.499,A -85,B 0,C 180,E1 2833.09,E2 2833.09} C_VEL
LIN {X 0,Y 607.884,Z 441.65,A -85,B 0,C 180,E1 2832.79,E2 2832.79} C_VEL
LIN {X 0,Y 607.887,Z 437.75,A -85,B 0,C 180,E1 2832.534,E2 2832.534} C_VEL
LIN {X 0,Y 607.897,Z 430.931,A -85,B 0,C 180,E1 2832.336,E2 2832.336} C_VEL
LIN {X 0,Y 607.904,Z 420.188,A -85,B 0,C 180,E1 2832.248,E2 2832.248} C_VEL
LIN {X 0,Y 607.905,Z 355.016,A -85,B 0,C 180,E1 2832.23,E2 2832.23} C_VEL
LIN {X 0,Y 607.903,Z 355.013,A -85,B 0,C 180,E1 2829.047,E2 2829.047} C_VEL
LIN {X 0,Y 607.891,Z 355.198,A -85,B 0,C 180,E1 2827.829,E2 2827.829} C_VEL
LIN {X 0,Y 607.902,Z 408.845,A -85,B 0,C 180,E1 2824.842,E2 2824.842} C_VEL
LIN {X 0,Y 607.881,Z 454.759,A -85,B 0,C 180,E1 2822.378,E2 2822.378} C_VEL
LIN {X 0,Y 607.913,Z 672.081,A -85,B 0,C 180,E1 2819.444,E2 2819.444} C_VEL
LIN {X 0,Y 607.899,Z 761.529,A -85,B 0,C 180,E1 2818.235,E2 2818.235} C_VEL
LIN {X 0,Y 607.909,Z 782.039,A -85,B 0,C 180,E1 2817.785,E2 2817.785} C_VEL
LIN {X 0,Y 607.907,Z 802.628,A -85,B 0,C 180,E1 2817.18,E2 2817.18} C_VEL
LIN {X 0,Y 607.903,Z 822.575,A -85,B 0,C 180,E1 2816.418,E2 2816.418} C_VEL
LIN {X 0,Y 607.918,Z 843.74,A -85,B 0,C 180,E1 2815.422,E2 2815.422} C_VEL
LIN {X 0,Y 607.916,Z 863.107,A -85,B 0,C 180,E1 2814.332,E2 2814.332} C_VEL
LIN {X 0,Y 607.915,Z 881.556,A -85,B 0,C 180,E1 2813.096,E2 2813.096} C_VEL
LIN {X 0,Y 607.911,Z 899.775,A -85,B 0,C 180,E1 2811.678,E2 2811.678} C_VEL
LIN {X 0,Y 607.913,Z 916.651,A -85,B 0,C 180,E1 2810.156,E2 2810.156} C_VEL
LIN {X 0,Y 607.918,Z 932.463,A -85,B 0,C 180,E1 2808.508,E2 2808.508} C_VEL
LIN {X 0,Y 607.918,Z 947.111,A -85,B 0,C 180,E1 2806.728,E2 2806.728} C_VEL
LIN {X 0,Y 607.915,Z 959.541,A -85,B 0,C 180,E1 2804.965,E2 2804.965} C_VEL
LIN {X 0,Y 607.917,Z 970.729,A -85,B 0,C 180,E1 2803.119,E2 2803.119} C_VEL
LIN {X 0,Y 607.903,Z 980.06,A -85,B 0,C 180,E1 2801.287,E2 2801.287} C_VEL
LIN {X 0,Y 607.896,Z 988.388,A -85,B 0,C 180,E1 2799.296,E2 2799.296} C_VEL
LIN {X 0,Y 607.891,Z 994.961,A -85,B 0,C 180,E1 2797.339,E2 2797.339} C_VEL
LIN {X 0,Y 607.9,Z 999.809,A -85,B 0,C 180,E1 2795.38,E2 2795.38} C_VEL
LIN {X 0,Y 607.913,Z 1003.346,A -85,B 0,C 180,E1 2793.29,E2 2793.29} C_VEL
LIN {X 0,Y 607.911,Z 1005.209,A -85,B 0,C 180,E1 2791.225,E2 2791.225} C_VEL
LIN {X 0,Y 607.895,Z 1005.329,A -85,B 0,C 180,E1 2789.246,E2 2789.246} C_VEL
LIN {X 0,Y 607.89,Z 1003.896,A -85,B 0,C 180,E1 2787.172,E2 2787.172} C_VEL
LIN {X 0,Y 607.896,Z 1000.987,A -85,B 0,C 180,E1 2785.188,E2 2785.188} C_VEL
LIN {X 0,Y 607.91,Z 996.4,A -85,B 0,C 180,E1 2783.199,E2 2783.199} C_VEL
LIN {X 0,Y 607.91,Z 990.239,A -85,B 0,C 180,E1 2781.202,E2 2781.202} C_VEL
LIN {X 0,Y 607.907,Z 982.658,A -85,B 0,C 180,E1 2779.289,E2 2779.289} C_VEL
LIN {X 0,Y 607.909,Z 973.328,A -85,B 0,C 180,E1 2777.365,E2 2777.365} C_VEL
LIN {X 0,Y 607.916,Z 962.747,A -85,B 0,C 180,E1 2775.523,E2 2775.523} C_VEL
LIN {X 0,Y 607.913,Z 950.036,A -85,B 0,C 180,E1 2773.665,E2 2773.665} C_VEL
LIN {X 0,Y 607.905,Z 935.869,A -85,B 0,C 180,E1 2771.889,E2 2771.889} C_VEL
LIN {X 0,Y 607.909,Z 920.096,A -85,B 0,C 180,E1 2770.185,E2 2770.185} C_VEL
LIN {X 0,Y 607.914,Z 903.502,A -85,B 0,C 180,E1 2768.635,E2 2768.635} C_VEL
LIN {X 0,Y 607.916,Z 885.139,A -85,B 0,C 180,E1 2767.16,E2 2767.16} C_VEL
LIN {X 0,Y 607.915,Z 866.679,A -85,B 0,C 180,E1 2765.898,E2 2765.898} C_VEL
LIN {X 0,Y 607.917,Z 846.558,A -85,B 0,C 180,E1 2764.726,E2 2764.726} C_VEL
LIN {X 0,Y 607.899,Z 826.382,A -85,B 0,C 180,E1 2763.74,E2 2763.74} C_VEL
LIN {X 0,Y 607.91,Z 805.509,A -85,B 0,C 180,E1 2762.923,E2 2762.923} C_VEL
LIN {X 0,Y 607.912,Z 783.805,A -85,B 0,C 180,E1 2762.26,E2 2762.26} C_VEL
LIN {X 0,Y 607.899,Z 763.078,A -85,B 0,C 180,E1 2761.793,E2 2761.793} C_VEL
LIN {X 0,Y 607.917,Z 720.893,A -85,B 0,C 180,E1 2761.203,E2 2761.203} C_VEL
LIN {X 0,Y 607.863,Z 490.978,A -85,B 0,C 180,E1 2758.116,E2 2758.116} C_VEL
LIN {X 0,Y 607.882,Z 454.241,A -85,B 0,C 180,E1 2757.602,E2 2757.602} C_VEL
LIN {X 0,Y 607.911,Z 399.078,A -85,B 0,C 180,E1 2754.623,E2 2754.623} C_VEL
LIN {X 0,Y 607.891,Z 355.015,A -85,B 0,C 180,E1 2752.157,E2 2752.157} C_VEL
LIN {X 0,Y 607.914,Z 355.014,A -85,B 0,C 180,E1 2748.986,E2 2748.986} C_VEL
LIN {X 0,Y 607.904,Z 355.016,A -85,B 0,C 180,E1 2747.753,E2 2747.753} C_VEL
LIN {X 0,Y 607.903,Z 425.086,A -85,B 0,C 180,E1 2747.733,E2 2747.733} C_VEL
LIN {X 0,Y 607.893,Z 434.04,A -85,B 0,C 180,E1 2747.595,E2 2747.595} C_VEL
LIN {X 0,Y 607.885,Z 439.038,A -85,B 0,C 180,E1 2747.402,E2 2747.402} C_VEL
LIN {X 0,Y 607.884,Z 441.863,A -85,B 0,C 180,E1 2747.188,E2 2747.188} C_VEL
LIN {X 0,Y 607.896,Z 443.499,A -85,B 0,C 180,E1 2746.91,E2 2746.91} C_VEL
LIN {X 0,Y 607.914,Z 443.592,A -85,B 0,C 180,E1 2746.496,E2 2746.496} C_VEL
LIN {X 0,Y 607.89,Z 441.764,A -85,B 0,C 180,E1 2746.044,E2 2746.044} C_VEL
LIN {X 0,Y 607.912,Z 437.097,A -85,B 0,C 180,E1 2745.466,E2 2745.466} C_VEL
LIN {X 0,Y 607.904,Z 428.655,A -85,B 0,C 180,E1 2744.745,E2 2744.745} C_VEL
LIN {X 0,Y 607.915,Z 409.979,A -85,B 0,C 180,E1 2743.562,E2 2743.562} C_VEL
LIN {X 0,Y 607.881,Z 370.359,A -85,B 0,C 180,E1 2741.068,E2 2741.068} C_VEL
LIN {X 0,Y 607.894,Z 355.012,A -85,B 0,C 180,E1 2740.045,E2 2740.045} C_VEL
LIN {X 0,Y 607.882,Z 355.013,A -85,B 0,C 180,E1 2736.929,E2 2736.929} C_VEL
LIN {X 0,Y 607.881,Z 355.013,A -85,B 0,C 180,E1 2733.776,E2 2733.776} C_VEL
LIN {X 0,Y 607.899,Z 355.012,A -85,B 0,C 180,E1 2730.656,E2 2730.656} C_VEL
LIN {X 0,Y 607.89,Z 355.015,A -85,B 0,C 180,E1 2727.528,E2 2727.528} C_VEL
LIN {X 0,Y 607.912,Z 355.013,A -85,B 0,C 180,E1 2724.382,E2 2724.382} C_VEL
LIN {X 0,Y 607.902,Z 355.015,A -85,B 0,C 180,E1 2721.159,E2 2721.159} C_VEL
LIN {X 0,Y 607.915,Z 355.013,A -85,B 0,C 180,E1 2717.912,E2 2717.912} C_VEL
LIN {X 0,Y 607.905,Z 355.015,A -85,B 0,C 180,E1 2714.672,E2 2714.672} C_VEL
LIN {X 0,Y 607.919,Z 355.014,A -85,B 0,C 180,E1 2711.479,E2 2711.479} C_VEL
LIN {X 0,Y 607.91,Z 355.015,A -85,B 0,C 180,E1 2708.227,E2 2708.227} C_VEL
LIN {X 0,Y 607.913,Z 355.015,A -85,B 0,C 180,E1 2705.001,E2 2705.001} C_VEL
LIN {X 0,Y 607.913,Z 355.016,A -85,B 0,C 180,E1 2701.791,E2 2701.791} C_VEL
LIN {X 0,Y 607.912,Z 355.015,A -85,B 0,C 180,E1 2698.586,E2 2698.586} C_VEL
LIN {X 0,Y 607.899,Z 355.014,A -85,B 0,C 180,E1 2696.736,E2 2696.736} C_VEL
LIN {X 0,Y 606.867,Z 355.139,A -85,B 0,C 180,E1 2696.01,E2 2696.01} C_VEL
LIN {X 0,Y 600.502,Z 355.939,A -85,B 0,C 180,E1 2693.973,E2 2693.973} C_VEL
LIN {X 0,Y 599.966,Z 356.002,A -85,B 0,C 180,E1 2693.443,E2 2693.443} C_VEL
LIN {X 0,Y 599.962,Z 356.004,A -85,B 0,C 180,E1 2690.31,E2 2690.31} C_VEL
LIN {X 0,Y 599.974,Z 356.003,A -85,B 0,C 180,E1 2687.096,E2 2687.096} C_VEL
LIN {X 0,Y 599.965,Z 356.004,A -85,B 0,C 180,E1 2683.84,E2 2683.84} C_VEL
LIN {X 0,Y 599.978,Z 356.002,A -85,B 0,C 180,E1 2680.601,E2 2680.601} C_VEL
LIN {X 0,Y 599.969,Z 356.003,A -85,B 0,C 180,E1 2677.358,E2 2677.358} C_VEL
LIN {X 0,Y 599.972,Z 356.003,A -85,B 0,C 180,E1 2674.111,E2 2674.111} C_VEL
LIN {X 0,Y 599.971,Z 356.003,A -85,B 0,C 180,E1 2670.838,E2 2670.838} C_VEL
LIN {X 0,Y 599.966,Z 356.004,A -85,B 0,C 180,E1 2667.659,E2 2667.659} C_VEL
LIN {X 0,Y 599.972,Z 356.001,A -85,B 0,C 180,E1 2664.436,E2 2664.436} C_VEL
LIN {X 0,Y 599.975,Z 356.004,A -85,B 0,C 180,E1 2661.2,E2 2661.2} C_VEL
LIN {X 0,Y 599.973,Z 356.002,A -85,B 0,C 180,E1 2657.938,E2 2657.938} C_VEL
LIN {X 0,Y 599.972,Z 356.004,A -85,B 0,C 180,E1 2654.689,E2 2654.689} C_VEL
LIN {X 0,Y 599.98,Z 356.003,A -85,B 0,C 180,E1 2651.416,E2 2651.416} C_VEL
LIN {X 0,Y 599.97,Z 356.003,A -85,B 0,C 180,E1 2648.131,E2 2648.131} C_VEL
LIN {X 0,Y 599.968,Z 356.004,A -85,B 0,C 180,E1 2644.922,E2 2644.922} C_VEL
LIN {X 0,Y 599.97,Z 356.005,A -85,B 0,C 180,E1 2641.777,E2 2641.777} C_VEL
LIN {X 0,Y 599.994,Z 356.211,A -85,B 0,C 180,E1 2640.453,E2 2640.453} C_VEL
LIN {X 0,Y 600.663,Z 358.734,A -85,B 0,C 180,E1 2640.24,E2 2640.24} C_VEL
LIN {X 0,Y 600.532,Z 404.092,A -85,B 0,C 180,E1 2637.142,E2 2637.142} C_VEL
LIN {X 0,Y 600.384,Z 450.964,A -85,B 0,C 180,E1 2634.028,E2 2634.028} C_VEL
LIN {X 0,Y 600.402,Z 473.538,A -85,B 0,C 180,E1 2632.575,E2 2632.575} C_VEL
LIN {X 0,Y 600.374,Z 683.005,A -85,B 0,C 180,E1 2629.915,E2 2629.915} C_VEL
LIN {X 0,Y 600.335,Z 702.108,A -85,B 0,C 180,E1 2629.485,E2 2629.485} C_VEL
LIN {X 0,Y 600.291,Z 720.108,A -85,B 0,C 180,E1 2628.901,E2 2628.901} C_VEL
LIN {X 0,Y 600.202,Z 737.679,A -85,B 0,C 180,E1 2628.15,E2 2628.15} C_VEL
LIN {X 0,Y 600.18,Z 754.381,A -85,B 0,C 180,E1 2627.249,E2 2627.249} C_VEL
LIN {X 0,Y 600.121,Z 770.212,A -85,B 0,C 180,E1 2626.205,E2 2626.205} C_VEL
LIN {X 0,Y 600.066,Z 785.12,A -85,B 0,C 180,E1 2625.017,E2 2625.017} C_VEL
LIN {X 0,Y 600.022,Z 799.03,A -85,B 0,C 180,E1 2623.687,E2 2623.687} C_VEL
LIN {X 0,Y 599.984,Z 811.832,A -85,B 0,C 180,E1 2622.218,E2 2622.218} C_VEL
LIN {X 0,Y 599.954,Z 823.073,A -85,B 0,C 180,E1 2620.66,E2 2620.66} C_VEL
LIN {X 0,Y 599.937,Z 832.77,A -85,B 0,C 180,E1 2619.013,E2 2619.013} C_VEL
LIN {X 0,Y 599.92,Z 840.492,A -85,B 0,C 180,E1 2617.373,E2 2617.373} C_VEL
LIN {X 0,Y 599.909,Z 846.77,A -85,B 0,C 180,E1 2615.643,E2 2615.643} C_VEL
LIN {X 0,Y 599.918,Z 851.277,A -85,B 0,C 180,E1 2613.918,E2 2613.918} C_VEL
LIN {X 0,Y 599.917,Z 854.235,A -85,B 0,C 180,E1 2612.101,E2 2612.101} C_VEL
LIN {X 0,Y 599.909,Z 855.429,A -85,B 0,C 180,E1 2610.286,E2 2610.286} C_VEL
LIN {X 0,Y 599.915,Z 854.879,A -85,B 0,C 180,E1 2608.472,E2 2608.472} C_VEL
LIN {X 0,Y 599.908,Z 852.578,A -85,B 0,C 180,E1 2606.656,E2 2606.656} C_VEL
LIN {X 0,Y 599.908,Z 848.714,A -85,B 0,C 180,E1 2604.932,E2 2604.932} C_VEL
LIN {X 0,Y 599.919,Z 843.132,A -85,B 0,C 180,E1 2603.204,E2 2603.204} C_VEL
LIN {X 0,Y 599.926,Z 835.678,A -85,B 0,C 180,E1 2601.47,E2 2601.47} C_VEL
LIN {X 0,Y 599.943,Z 826.701,A -85,B 0,C 180,E1 2599.825,E2 2599.825} C_VEL
LIN {X 0,Y 599.969,Z 816.266,A -85,B 0,C 180,E1 2598.269,E2 2598.269} C_VEL
LIN {X 0,Y 600.004,Z 804.389,A -85,B 0,C 180,E1 2596.803,E2 2596.803} C_VEL
LIN {X 0,Y 600.051,Z 791.04,A -85,B 0,C 180,E1 2595.427,E2 2595.427} C_VEL
LIN {X 0,Y 600.107,Z 776.019,A -85,B 0,C 180,E1 2594.142,E2 2594.142} C_VEL
LIN {X 0,Y 600.164,Z 760.628,A -85,B 0,C 180,E1 2593.049,E2 2593.049} C_VEL
LIN {X 0,Y 600.192,Z 744.408,A -85,B 0,C 180,E1 2592.1,E2 2592.1} C_VEL
LIN {X 0,Y 600.264,Z 727.309,A -85,B 0,C 180,E1 2591.294,E2 2591.294} C_VEL
LIN {X 0,Y 600.325,Z 708.782,A -85,B 0,C 180,E1 2590.621,E2 2590.621} C_VEL
LIN {X 0,Y 600.365,Z 689.701,A -85,B 0,C 180,E1 2590.126,E2 2590.126} C_VEL
LIN {X 0,Y 600.387,Z 669.129,A -85,B 0,C 180,E1 2589.796,E2 2589.796} C_VEL
LIN {X 0,Y 600.341,Z 473.074,A -85,B 0,C 180,E1 2587.326,E2 2587.326} C_VEL
LIN {X 0,Y 600.457,Z 425.294,A -85,B 0,C 180,E1 2584.186,E2 2584.186} C_VEL
LIN {X 0,Y 600.609,Z 379.26,A -85,B 0,C 180,E1 2581.084,E2 2581.084} C_VEL
LIN {X 0,Y 600.45,Z 357.981,A -85,B 0,C 180,E1 2579.606,E2 2579.606} C_VEL
LIN {X 0,Y 599.961,Z 356.006,A -85,B 0,C 180,E1 2579.422,E2 2579.422} C_VEL
LIN {X 0,Y 599.918,Z 356.001,A -85,B 0,C 180,E1 2576.27,E2 2576.27} C_VEL
LIN {X 0,Y 599.958,Z 356.004,A -85,B 0,C 180,E1 2573.252,E2 2573.252} C_VEL
LIN {X 0,Y 599.916,Z 356,A -85,B 0,C 180,E1 2570.056,E2 2570.056} C_VEL
LIN {X 0,Y 599.944,Z 356.003,A -85,B 0,C 180,E1 2567.158,E2 2567.158} C_VEL
LIN {X 0,Y 599.917,Z 356,A -85,B 0,C 180,E1 2563.895,E2 2563.895} C_VEL
LIN {X 0,Y 599.946,Z 356.003,A -85,B 0,C 180,E1 2560.917,E2 2560.917} C_VEL
LIN {X 0,Y 599.917,Z 356.001,A -85,B 0,C 180,E1 2557.658,E2 2557.658} C_VEL
LIN {X 0,Y 599.954,Z 356.005,A -85,B 0,C 180,E1 2554.632,E2 2554.632} C_VEL
LIN {X 0,Y 599.988,Z 356.088,A -85,B 0,C 180,E1 2552.312,E2 2552.312} C_VEL
LIN {X 0,Y 600.779,Z 359.302,A -85,B 0,C 180,E1 2552.01,E2 2552.01} C_VEL
LIN {X 0,Y 600.591,Z 396.084,A -85,B 0,C 180,E1 2549.266,E2 2549.266} C_VEL
LIN {X 0,Y 600.471,Z 439.76,A -85,B 0,C 180,E1 2546.137,E2 2546.137} C_VEL
LIN {X 0,Y 600.335,Z 485.828,A -85,B 0,C 180,E1 2542.923,E2 2542.923} C_VEL
LIN {X 0,Y 600.231,Z 532.899,A -85,B 0,C 180,E1 2539.714,E2 2539.714} C_VEL
LIN {X 0,Y 600.13,Z 580.944,A -85,B 0,C 180,E1 2536.503,E2 2536.503} C_VEL
LIN {X 0,Y 600.17,Z 588.969,A -85,B 0,C 180,E1 2535.999,E2 2535.999} C_VEL
LIN {X 0,Y 600.134,Z 731.702,A -85,B 0,C 180,E1 2534.241,E2 2534.241} C_VEL
LIN {X 0,Y 600.118,Z 748.908,A -85,B 0,C 180,E1 2533.833,E2 2533.833} C_VEL
LIN {X 0,Y 600.086,Z 763.987,A -85,B 0,C 180,E1 2533.293,E2 2533.293} C_VEL
LIN {X 0,Y 600.057,Z 779.133,A -85,B 0,C 180,E1 2532.56,E2 2532.56} C_VEL
LIN {X 0,Y 600.025,Z 793.17,A -85,B 0,C 180,E1 2531.681,E2 2531.681} C_VEL
LIN {X 0,Y 599.995,Z 806.097,A -85,B 0,C 180,E1 2530.66,E2 2530.66} C_VEL
LIN {X 0,Y 599.966,Z 817.936,A -85,B 0,C 180,E1 2529.497,E2 2529.497} C_VEL
LIN {X 0,Y 599.944,Z 828.147,A -85,B 0,C 180,E1 2528.241,E2 2528.241} C_VEL
LIN {X 0,Y 599.931,Z 836.904,A -85,B 0,C 180,E1 2526.892,E2 2526.892} C_VEL
LIN {X 0,Y 599.919,Z 844.062,A -85,B 0,C 180,E1 2525.452,E2 2525.452} C_VEL
LIN {X 0,Y 599.915,Z 849.654,A -85,B 0,C 180,E1 2523.919,E2 2523.919} C_VEL
LIN {X 0,Y 599.914,Z 853.305,A -85,B 0,C 180,E1 2522.388,E2 2522.388} C_VEL
LIN {X 0,Y 599.913,Z 855.234,A -85,B 0,C 180,E1 2520.764,E2 2520.764} C_VEL
LIN {X 0,Y 599.913,Z 855.297,A -85,B 0,C 180,E1 2519.236,E2 2519.236} C_VEL
LIN {X 0,Y 599.914,Z 853.454,A -85,B 0,C 180,E1 2517.612,E2 2517.612} C_VEL
LIN {X 0,Y 599.915,Z 849.938,A -85,B 0,C 180,E1 2516.082,E2 2516.082} C_VEL
LIN {X 0,Y 599.919,Z 844.443,A -85,B 0,C 180,E1 2514.549,E2 2514.549} C_VEL
LIN {X 0,Y 599.927,Z 837.406,A -85,B 0,C 180,E1 2513.108,E2 2513.108} C_VEL
LIN {X 0,Y 599.944,Z 828.808,A -85,B 0,C 180,E1 2511.76,E2 2511.76} C_VEL
LIN {X 0,Y 599.962,Z 818.731,A -85,B 0,C 180,E1 2510.504,E2 2510.504} C_VEL
LIN {X 0,Y 599.992,Z 807.126,A -85,B 0,C 180,E1 2509.341,E2 2509.341} C_VEL
LIN {X 0,Y 600.024,Z 793.757,A -85,B 0,C 180,E1 2508.27,E2 2508.27} C_VEL
LIN {X 0,Y 600.054,Z 779.892,A -85,B 0,C 180,E1 2507.392,E2 2507.392} C_VEL
LIN {X 0,Y 600.086,Z 764.549,A -85,B 0,C 180,E1 2506.64,E2 2506.64} C_VEL
LIN {X 0,Y 600.114,Z 748.939,A -85,B 0,C 180,E1 2506.078,E2 2506.078} C_VEL
LIN {X 0,Y 600.132,Z 731.323,A -85,B 0,C 180,E1 2505.661,E2 2505.661} C_VEL
LIN {X 0,Y 600.11,Z 588.31,A -85,B 0,C 180,E1 2503.895,E2 2503.895} C_VEL
LIN {X 0,Y 600.207,Z 541,A -85,B 0,C 180,E1 2500.741,E2 2500.741} C_VEL
LIN {X 0,Y 600.309,Z 494.426,A -85,B 0,C 180,E1 2497.578,E2 2497.578} C_VEL
LIN {X 0,Y 600.436,Z 450.021,A -85,B 0,C 180,E1 2494.496,E2 2494.496} C_VEL
LIN {X 0,Y 600.565,Z 405.065,A -85,B 0,C 180,E1 2491.295,E2 2491.295} C_VEL
LIN {X 0,Y 600.736,Z 395.904,A -85,B 0,C 180,E1 2490.594,E2 2490.594} C_VEL
LIN {X 0,Y 601.919,Z 378.174,A -85,B 0,C 180,E1 2489.062,E2 2489.062} C_VEL
LIN {X 0,Y 602.095,Z 360.548,A -85,B 0,C 180,E1 2487.307,E2 2487.307} C_VEL
LIN {X 0,Y 600.329,Z 357.617,A -85,B 0,C 180,E1 2486.73,E2 2486.73} C_VEL
LIN {X 0,Y 599.977,Z 356.003,A -85,B 0,C 180,E1 2486.474,E2 2486.474} C_VEL
LIN {X 0,Y 599.96,Z 356.005,A -85,B 0,C 180,E1 2483.253,E2 2483.253} C_VEL
LIN {X 0,Y 599.972,Z 356.003,A -85,B 0,C 180,E1 2480.05,E2 2480.05} C_VEL
LIN {X 0,Y 599.995,Z 356.131,A -85,B 0,C 180,E1 2479.679,E2 2479.679} C_VEL
LIN {X 0,Y 601.224,Z 359.496,A -85,B 0,C 180,E1 2479.377,E2 2479.377} C_VEL
LIN {X 0,Y 600.818,Z 396.645,A -85,B 0,C 180,E1 2477.438,E2 2477.438} C_VEL
LIN {X 0,Y 601.215,Z 425.807,A -85,B 0,C 180,E1 2475.96,E2 2475.96} C_VEL
LIN {X 0,Y 602.192,Z 437,A -85,B 0,C 180,E1 2475.287,E2 2475.287} C_VEL
LIN {X 0,Y 603.27,Z 444.663,A -85,B 0,C 180,E1 2474.647,E2 2474.647} C_VEL
LIN {X 0,Y 604.218,Z 448.984,A -85,B 0,C 180,E1 2474.096,E2 2474.096} C_VEL
LIN {X 0,Y 605.049,Z 451.053,A -85,B 0,C 180,E1 2473.56,E2 2473.56} C_VEL
LIN {X 0,Y 605.499,Z 451.21,A -85,B 0,C 180,E1 2473.048,E2 2473.048} C_VEL
LIN {X 0,Y 605.49,Z 449.534,A -85,B 0,C 180,E1 2472.596,E2 2472.596} C_VEL
LIN {X 0,Y 605.017,Z 445.99,A -85,B 0,C 180,E1 2472.206,E2 2472.206} C_VEL
LIN {X 0,Y 604.191,Z 440.551,A -85,B 0,C 180,E1 2471.917,E2 2471.917} C_VEL
LIN {X 0,Y 603.167,Z 432.831,A -85,B 0,C 180,E1 2471.75,E2 2471.75} C_VEL
LIN {X 0,Y 602.559,Z 420.495,A -85,B 0,C 180,E1 2471.685,E2 2471.685} C_VEL
LIN {X 0,Y 602.544,Z 360.947,A -85,B 0,C 180,E1 2471.683,E2 2471.683} C_VEL
LIN {X 0,Y 600.553,Z 358.143,A -85,B 0,C 180,E1 2471.469,E2 2471.469} C_VEL
LIN {X 0,Y 599.98,Z 356.001,A -85,B 0,C 180,E1 2471.39,E2 2471.39} C_VEL
LIN {X 0,Y 599.983,Z 356.11,A -85,B 0,C 180,E1 2468.365,E2 2468.365} C_VEL
LIN {X 0,Y 601.234,Z 359.87,A -85,B 0,C 180,E1 2468.054,E2 2468.054} C_VEL
LIN {X 0,Y 601.052,Z 412.933,A -85,B 0,C 180,E1 2465.071,E2 2465.071} C_VEL
LIN {X 0,Y 601.009,Z 455.268,A -85,B 0,C 180,E1 2462.787,E2 2462.787} C_VEL
LIN {X 0,Y 600.95,Z 625.941,A -85,B 0,C 180,E1 2460.444,E2 2460.444} C_VEL
LIN {X 0,Y 600.844,Z 761.335,A -85,B 0,C 180,E1 2458.6,E2 2458.6} C_VEL
LIN {X 0,Y 600.79,Z 782.629,A -85,B 0,C 180,E1 2458.129,E2 2458.129} C_VEL
LIN {X 0,Y 600.704,Z 804.075,A -85,B 0,C 180,E1 2457.481,E2 2457.481} C_VEL
LIN {X 0,Y 600.625,Z 825.259,A -85,B 0,C 180,E1 2456.651,E2 2456.651} C_VEL
LIN {X 0,Y 600.538,Z 844.74,A -85,B 0,C 180,E1 2455.704,E2 2455.704} C_VEL
LIN {X 0,Y 600.435,Z 863.923,A -85,B 0,C 180,E1 2454.602,E2 2454.602} C_VEL
LIN {X 0,Y 600.349,Z 883.012,A -85,B 0,C 180,E1 2453.3,E2 2453.3} C_VEL
LIN {X 0,Y 600.246,Z 900.553,A -85,B 0,C 180,E1 2451.903,E2 2451.903} C_VEL
LIN {X 0,Y 600.159,Z 918.174,A -85,B 0,C 180,E1 2450.275,E2 2450.275} C_VEL
LIN {X 0,Y 600.093,Z 933.317,A -85,B 0,C 180,E1 2448.658,E2 2448.658} C_VEL
LIN {X 0,Y 600.043,Z 947.883,A -85,B 0,C 180,E1 2446.855,E2 2446.855} C_VEL
LIN {X 0,Y 599.996,Z 960.186,A -85,B 0,C 180,E1 2445.068,E2 2445.068} C_VEL
LIN {X 0,Y 599.958,Z 971.77,A -85,B 0,C 180,E1 2443.1,E2 2443.1} C_VEL
LIN {X 0,Y 599.937,Z 981.429,A -85,B 0,C 180,E1 2441.147,E2 2441.147} C_VEL
LIN {X 0,Y 599.912,Z 989.175,A -85,B 0,C 180,E1 2439.207,E2 2439.207} C_VEL
LIN {X 0,Y 599.899,Z 995.893,A -85,B 0,C 180,E1 2437.085,E2 2437.085} C_VEL
LIN {X 0,Y 599.893,Z 1000.428,A -85,B 0,C 180,E1 2435.164,E2 2435.164} C_VEL
LIN {X 0,Y 599.902,Z 1003.562,A -85,B 0,C 180,E1 2433.153,E2 2433.153} C_VEL
LIN {X 0,Y 599.917,Z 1005.239,A -85,B 0,C 180,E1 2431.146,E2 2431.146} C_VEL
LIN {X 0,Y 599.899,Z 1005.31,A -85,B 0,C 180,E1 2429.141,E2 2429.141} C_VEL
LIN {X 0,Y 599.893,Z 1003.787,A -85,B 0,C 180,E1 2427.039,E2 2427.039} C_VEL
LIN {X 0,Y 599.892,Z 1000.825,A -85,B 0,C 180,E1 2425.028,E2 2425.028} C_VEL
LIN {X 0,Y 599.904,Z 996.149,A -85,B 0,C 180,E1 2423.012,E2 2423.012} C_VEL
LIN {X 0,Y 599.918,Z 989.532,A -85,B 0,C 180,E1 2420.89,E2 2420.89} C_VEL
LIN {X 0,Y 599.936,Z 981.847,A -85,B 0,C 180,E1 2418.951,E2 2418.951} C_VEL
LIN {X 0,Y 599.953,Z 972.293,A -85,B 0,C 180,E1 2416.998,E2 2416.998} C_VEL
LIN {X 0,Y 599.991,Z 960.831,A -85,B 0,C 180,E1 2415.031,E2 2415.031} C_VEL
LIN {X 0,Y 600.037,Z 948.623,A -85,B 0,C 180,E1 2413.246,E2 2413.246} C_VEL
LIN {X 0,Y 600.087,Z 934.241,A -85,B 0,C 180,E1 2411.452,E2 2411.452} C_VEL
LIN {X 0,Y 600.16,Z 918.686,A -85,B 0,C 180,E1 2409.776,E2 2409.776} C_VEL
LIN {X 0,Y 600.244,Z 901.697,A -85,B 0,C 180,E1 2408.194,E2 2408.194} C_VEL
LIN {X 0,Y 600.347,Z 883.747,A -85,B 0,C 180,E1 2406.752,E2 2406.752} C_VEL
LIN {X 0,Y 600.428,Z 864.734,A -85,B 0,C 180,E1 2405.451,E2 2405.451} C_VEL
LIN {X 0,Y 600.536,Z 845.746,A -85,B 0,C 180,E1 2404.349,E2 2404.349} C_VEL
LIN {X 0,Y 600.621,Z 825.82,A -85,B 0,C 180,E1 2403.373,E2 2403.373} C_VEL
LIN {X 0,Y 600.703,Z 804.787,A -85,B 0,C 180,E1 2402.545,E2 2402.545} C_VEL
LIN {X 0,Y 600.79,Z 783.016,A -85,B 0,C 180,E1 2401.881,E2 2401.881} C_VEL
LIN {X 0,Y 600.843,Z 761.694,A -85,B 0,C 180,E1 2401.406,E2 2401.406} C_VEL
LIN {X 0,Y 600.953,Z 664.686,A -85,B 0,C 180,E1 2400.081,E2 2400.081} C_VEL
LIN {X 0,Y 601.106,Z 455.877,A -85,B 0,C 180,E1 2397.227,E2 2397.227} C_VEL
LIN {X 0,Y 600.91,Z 453.716,A -85,B 0,C 180,E1 2397.151,E2 2397.151} C_VEL
LIN {X 0,Y 601.107,Z 399.078,A -85,B 0,C 180,E1 2394.162,E2 2394.162} C_VEL
LIN {X 0,Y 601.185,Z 359.366,A -85,B 0,C 180,E1 2391.913,E2 2391.913} C_VEL
LIN {X 0,Y 599.972,Z 356.004,A -85,B 0,C 180,E1 2391.6,E2 2391.6} C_VEL
LIN {X 0,Y 600.011,Z 356.228,A -85,B 0,C 180,E1 2388.589,E2 2388.589} C_VEL
LIN {X 0,Y 601.129,Z 359.253,A -85,B 0,C 180,E1 2388.469,E2 2388.469} C_VEL
LIN {X 0,Y 602.553,Z 360.956,A -85,B 0,C 180,E1 2388.316,E2 2388.316} C_VEL
LIN {X 0,Y 602.742,Z 427.328,A -85,B 0,C 180,E1 2388.296,E2 2388.296} C_VEL
LIN {X 0,Y 603.736,Z 437.341,A -85,B 0,C 180,E1 2388.176,E2 2388.176} C_VEL
LIN {X 0,Y 604.657,Z 443.609,A -85,B 0,C 180,E1 2387.947,E2 2387.947} C_VEL
LIN {X 0,Y 605.289,Z 447.836,A -85,B 0,C 180,E1 2387.627,E2 2387.627} C_VEL
LIN {X 0,Y 605.55,Z 450.423,A -85,B 0,C 180,E1 2387.228,E2 2387.228} C_VEL
LIN {X 0,Y 605.374,Z 451.366,A -85,B 0,C 180,E1 2386.75,E2 2386.75} C_VEL
LIN {X 0,Y 604.79,Z 450.583,A -85,B 0,C 180,E1 2386.258,E2 2386.258} C_VEL
LIN {X 0,Y 603.918,Z 447.856,A -85,B 0,C 180,E1 2385.729,E2 2385.729} C_VEL
LIN {X 0,Y 602.926,Z 442.514,A -85,B 0,C 180,E1 2385.149,E2 2385.149} C_VEL
LIN {X 0,Y 601.846,Z 433.101,A -85,B 0,C 180,E1 2384.446,E2 2384.446} C_VEL
LIN {X 0,Y 601.733,Z 378.728,A -85,B 0,C 180,E1 2381.021,E2 2381.021} C_VEL
LIN {X 0,Y 601.805,Z 360.211,A -85,B 0,C 180,E1 2379.797,E2 2379.797} C_VEL
LIN {X 0,Y 600.136,Z 356.963,A -85,B 0,C 180,E1 2379.402,E2 2379.402} C_VEL
LIN {X 0,Y 599.964,Z 356.004,A -85,B 0,C 180,E1 2379.292,E2 2379.292} C_VEL
LIN {X 0,Y 599.979,Z 356.003,A -85,B 0,C 180,E1 2376.034,E2 2376.034} C_VEL
LIN {X 0,Y 599.961,Z 356.002,A -85,B 0,C 180,E1 2372.794,E2 2372.794} C_VEL
LIN {X 0,Y 599.975,Z 356.002,A -85,B 0,C 180,E1 2369.552,E2 2369.552} C_VEL
LIN {X 0,Y 599.957,Z 356.004,A -85,B 0,C 180,E1 2366.314,E2 2366.314} C_VEL
LIN {X 0,Y 599.969,Z 356.003,A -85,B 0,C 180,E1 2363.056,E2 2363.056} C_VEL
LIN {X 0,Y 599.952,Z 356.004,A -85,B 0,C 180,E1 2359.875,E2 2359.875} C_VEL
LIN {X 0,Y 599.954,Z 356.002,A -85,B 0,C 180,E1 2356.757,E2 2356.757} C_VEL
LIN {X 0,Y 599.965,Z 356,A -85,B 0,C 180,E1 2353.59,E2 2353.59} C_VEL
LIN {X 0,Y 599.939,Z 356.003,A -85,B 0,C 180,E1 2350.369,E2 2350.369} C_VEL
LIN {X 0,Y 599.975,Z 355.999,A -85,B 0,C 180,E1 2347.084,E2 2347.084} C_VEL
LIN {X 0,Y 599.93,Z 356.004,A -85,B 0,C 180,E1 2343.918,E2 2343.918} C_VEL
LIN {X 0,Y 599.966,Z 356,A -85,B 0,C 180,E1 2340.668,E2 2340.668} C_VEL
LIN {X 0,Y 599.923,Z 356.004,A -85,B 0,C 180,E1 2337.612,E2 2337.612} C_VEL
LIN {X 0,Y 599.952,Z 356,A -85,B 0,C 180,E1 2334.357,E2 2334.357} C_VEL
LIN {X 0,Y 599.966,Z 356.002,A -85,B 0,C 180,E1 2333.443,E2 2333.443} C_VEL
LIN {X 0,Y 598.97,Z 356.123,A -85,B 0,C 180,E1 2332.708,E2 2332.708} C_VEL
LIN {X 0,Y 592.467,Z 356.939,A -85,B 0,C 180,E1 2330.591,E2 2330.591} C_VEL
LIN {X 0,Y 592.002,Z 356.993,A -85,B 0,C 180,E1 2330.107,E2 2330.107} C_VEL
LIN {X 0,Y 592.034,Z 356.99,A -85,B 0,C 180,E1 2326.92,E2 2326.92} C_VEL
LIN {X 0,Y 592.014,Z 356.993,A -85,B 0,C 180,E1 2323.718,E2 2323.718} C_VEL
LIN {X 0,Y 592.04,Z 356.989,A -85,B 0,C 180,E1 2320.453,E2 2320.453} C_VEL
LIN {X 0,Y 592.015,Z 356.991,A -85,B 0,C 180,E1 2317.142,E2 2317.142} C_VEL
LIN {X 0,Y 592.019,Z 356.991,A -85,B 0,C 180,E1 2313.952,E2 2313.952} C_VEL
LIN {X 0,Y 592.029,Z 356.991,A -85,B 0,C 180,E1 2310.785,E2 2310.785} C_VEL
LIN {X 0,Y 592.015,Z 356.993,A -85,B 0,C 180,E1 2307.515,E2 2307.515} C_VEL
LIN {X 0,Y 592.034,Z 356.987,A -85,B 0,C 180,E1 2304.325,E2 2304.325} C_VEL
LIN {X 0,Y 592.02,Z 356.993,A -85,B 0,C 180,E1 2301.077,E2 2301.077} C_VEL
LIN {X 0,Y 592.036,Z 356.989,A -85,B 0,C 180,E1 2297.851,E2 2297.851} C_VEL
LIN {X 0,Y 592.029,Z 356.992,A -85,B 0,C 180,E1 2294.633,E2 2294.633} C_VEL
LIN {X 0,Y 592.04,Z 356.992,A -85,B 0,C 180,E1 2291.423,E2 2291.423} C_VEL
LIN {X 0,Y 592.035,Z 356.992,A -85,B 0,C 180,E1 2288.179,E2 2288.179} C_VEL
LIN {X 0,Y 592.03,Z 356.994,A -85,B 0,C 180,E1 2284.926,E2 2284.926} C_VEL
LIN {X 0,Y 592.035,Z 356.993,A -85,B 0,C 180,E1 2281.659,E2 2281.659} C_VEL
LIN {X 0,Y 592.065,Z 357.236,A -85,B 0,C 180,E1 2280.833,E2 2280.833} C_VEL
LIN {X 0,Y 593.42,Z 362.001,A -85,B 0,C 180,E1 2280.418,E2 2280.418} C_VEL
LIN {X 0,Y 593.151,Z 407.281,A -85,B 0,C 180,E1 2277.29,E2 2277.29} C_VEL
LIN {X 0,Y 592.872,Z 453.8,A -85,B 0,C 180,E1 2274.163,E2 2274.163} C_VEL
LIN {X 0,Y 592.856,Z 473.576,A -85,B 0,C 180,E1 2272.878,E2 2272.878} C_VEL
LIN {X 0,Y 593.105,Z 487.374,A -85,B 0,C 180,E1 2272.691,E2 2272.691} C_VEL
LIN {X 0,Y 592.849,Z 682.848,A -85,B 0,C 180,E1 2270.182,E2 2270.182} C_VEL
LIN {X 0,Y 592.774,Z 701.969,A -85,B 0,C 180,E1 2269.749,E2 2269.749} C_VEL
LIN {X 0,Y 592.676,Z 720.549,A -85,B 0,C 180,E1 2269.137,E2 2269.137} C_VEL
LIN {X 0,Y 592.538,Z 737.697,A -85,B 0,C 180,E1 2268.394,E2 2268.394} C_VEL
LIN {X 0,Y 592.458,Z 754.395,A -85,B 0,C 180,E1 2267.481,E2 2267.481} C_VEL
LIN {X 0,Y 592.331,Z 770.884,A -85,B 0,C 180,E1 2266.373,E2 2266.373} C_VEL
LIN {X 0,Y 592.217,Z 786.233,A -85,B 0,C 180,E1 2265.12,E2 2265.12} C_VEL
LIN {X 0,Y 592.128,Z 799.965,A -85,B 0,C 180,E1 2263.774,E2 2263.774} C_VEL
LIN {X 0,Y 592.053,Z 812.615,A -85,B 0,C 180,E1 2262.286,E2 2262.286} C_VEL
LIN {X 0,Y 591.996,Z 823.719,A -85,B 0,C 180,E1 2260.707,E2 2260.707} C_VEL
LIN {X 0,Y 591.959,Z 833.293,A -85,B 0,C 180,E1 2259.037,E2 2259.037} C_VEL
LIN {X 0,Y 591.93,Z 840.901,A -85,B 0,C 180,E1 2257.375,E2 2257.375} C_VEL
LIN {X 0,Y 591.913,Z 847.075,A -85,B 0,C 180,E1 2255.622,E2 2255.622} C_VEL
LIN {X 0,Y 591.918,Z 851.483,A -85,B 0,C 180,E1 2253.874,E2 2253.874} C_VEL
LIN {X 0,Y 591.916,Z 854.348,A -85,B 0,C 180,E1 2252.033,E2 2252.033} C_VEL
LIN {X 0,Y 591.911,Z 855.452,A -85,B 0,C 180,E1 2250.193,E2 2250.193} C_VEL
LIN {X 0,Y 591.914,Z 854.813,A -85,B 0,C 180,E1 2248.354,E2 2248.354} C_VEL
LIN {X 0,Y 591.907,Z 852.42,A -85,B 0,C 180,E1 2246.513,E2 2246.513} C_VEL
LIN {X 0,Y 591.913,Z 848.46,A -85,B 0,C 180,E1 2244.766,E2 2244.766} C_VEL
LIN {X 0,Y 591.928,Z 842.778,A -85,B 0,C 180,E1 2243.014,E2 2243.014} C_VEL
LIN {X 0,Y 591.94,Z 835.677,A -85,B 0,C 180,E1 2241.354,E2 2241.354} C_VEL
LIN {X 0,Y 591.979,Z 826.7,A -85,B 0,C 180,E1 2239.686,E2 2239.686} C_VEL
LIN {X 0,Y 592.026,Z 816.265,A -85,B 0,C 180,E1 2238.109,E2 2238.109} C_VEL
LIN {X 0,Y 592.105,Z 803.96,A -85,B 0,C 180,E1 2236.573,E2 2236.573} C_VEL
LIN {X 0,Y 592.201,Z 790.51,A -85,B 0,C 180,E1 2235.179,E2 2235.179} C_VEL
LIN {X 0,Y 592.303,Z 776.009,A -85,B 0,C 180,E1 2233.928,E2 2233.928} C_VEL
LIN {X 0,Y 592.418,Z 760.28,A -85,B 0,C 180,E1 2232.799,E2 2232.799} C_VEL
LIN {X 0,Y 592.506,Z 743.415,A -85,B 0,C 180,E1 2231.808,E2 2231.808} C_VEL
LIN {X 0,Y 592.643,Z 726.142,A -85,B 0,C 180,E1 2230.997,E2 2230.997} C_VEL
LIN {X 0,Y 592.753,Z 707.395,A -85,B 0,C 180,E1 2230.322,E2 2230.322} C_VEL
LIN {X 0,Y 592.832,Z 688.391,A -85,B 0,C 180,E1 2229.837,E2 2229.837} C_VEL
LIN {X 0,Y 592.879,Z 666.66,A -85,B 0,C 180,E1 2229.498,E2 2229.498} C_VEL
LIN {X 0,Y 592.955,Z 474.197,A -85,B 0,C 180,E1 2227.044,E2 2227.044} C_VEL
LIN {X 0,Y 592.796,Z 472.189,A -85,B 0,C 180,E1 2226.964,E2 2226.964} C_VEL
LIN {X 0,Y 593.028,Z 425.284,A -85,B 0,C 180,E1 2223.839,E2 2223.839} C_VEL
LIN {X 0,Y 593.327,Z 379.17,A -85,B 0,C 180,E1 2220.689,E2 2220.689} C_VEL
LIN {X 0,Y 593.226,Z 360.883,A -85,B 0,C 180,E1 2219.402,E2 2219.402} C_VEL
LIN {X 0,Y 592.037,Z 356.991,A -85,B 0,C 180,E1 2219.042,E2 2219.042} C_VEL
LIN {X 0,Y 591.974,Z 356.991,A -85,B 0,C 180,E1 2216.008,E2 2216.008} C_VEL
LIN {X 0,Y 592.038,Z 356.989,A -85,B 0,C 180,E1 2212.858,E2 2212.858} C_VEL
LIN {X 0,Y 591.973,Z 356.99,A -85,B 0,C 180,E1 2209.769,E2 2209.769} C_VEL
LIN {X 0,Y 592.04,Z 356.988,A -85,B 0,C 180,E1 2206.71,E2 2206.71} C_VEL
LIN {X 0,Y 591.973,Z 356.99,A -85,B 0,C 180,E1 2203.695,E2 2203.695} C_VEL
LIN {X 0,Y 592.041,Z 356.991,A -85,B 0,C 180,E1 2200.537,E2 2200.537} C_VEL
LIN {X 0,Y 591.972,Z 356.991,A -85,B 0,C 180,E1 2197.449,E2 2197.449} C_VEL
LIN {X 0,Y 592.038,Z 356.989,A -85,B 0,C 180,E1 2194.325,E2 2194.325} C_VEL
LIN {X 0,Y 592.011,Z 357.114,A -85,B 0,C 180,E1 2192.759,E2 2192.759} C_VEL
LIN {X 0,Y 593.731,Z 362.844,A -85,B 0,C 180,E1 2192.208,E2 2192.208} C_VEL
LIN {X 0,Y 593.313,Z 399.869,A -85,B 0,C 180,E1 2189.394,E2 2189.394} C_VEL
LIN {X 0,Y 593.025,Z 442.922,A -85,B 0,C 180,E1 2186.264,E2 2186.264} C_VEL
LIN {X 0,Y 592.767,Z 487.877,A -85,B 0,C 180,E1 2183.09,E2 2183.09} C_VEL
LIN {X 0,Y 592.555,Z 534.411,A -85,B 0,C 180,E1 2179.877,E2 2179.877} C_VEL
LIN {X 0,Y 592.356,Z 582.448,A -85,B 0,C 180,E1 2176.625,E2 2176.625} C_VEL
LIN {X 0,Y 592.393,Z 589.008,A -85,B 0,C 180,E1 2176.215,E2 2176.215} C_VEL
LIN {X 0,Y 592.376,Z 731.747,A -85,B 0,C 180,E1 2174.432,E2 2174.432} C_VEL
LIN {X 0,Y 592.337,Z 748.935,A -85,B 0,C 180,E1 2174.018,E2 2174.018} C_VEL
LIN {X 0,Y 592.272,Z 763.977,A -85,B 0,C 180,E1 2173.472,E2 2173.472} C_VEL
LIN {X 0,Y 592.209,Z 779.151,A -85,B 0,C 180,E1 2172.729,E2 2172.729} C_VEL
LIN {X 0,Y 592.14,Z 793.163,A -85,B 0,C 180,E1 2171.839,E2 2171.839} C_VEL
LIN {X 0,Y 592.074,Z 806.108,A -85,B 0,C 180,E1 2170.804,E2 2170.804} C_VEL
LIN {X 0,Y 592.017,Z 817.933,A -85,B 0,C 180,E1 2169.625,E2 2169.625} C_VEL
LIN {X 0,Y 591.972,Z 828.15,A -85,B 0,C 180,E1 2168.352,E2 2168.352} C_VEL
LIN {X 0,Y 591.946,Z 836.908,A -85,B 0,C 180,E1 2166.986,E2 2166.986} C_VEL
LIN {X 0,Y 591.925,Z 844.061,A -85,B 0,C 180,E1 2165.525,E2 2165.525} C_VEL
LIN {X 0,Y 591.917,Z 849.657,A -85,B 0,C 180,E1 2163.972,E2 2163.972} C_VEL
LIN {X 0,Y 591.915,Z 853.3,A -85,B 0,C 180,E1 2162.421,E2 2162.421} C_VEL
LIN {X 0,Y 591.915,Z 855.167,A -85,B 0,C 180,E1 2160.871,E2 2160.871} C_VEL
LIN {X 0,Y 591.913,Z 855.357,A -85,B 0,C 180,E1 2159.323,E2 2159.323} C_VEL
LIN {X 0,Y 591.916,Z 853.761,A -85,B 0,C 180,E1 2157.774,E2 2157.774} C_VEL
LIN {X 0,Y 591.917,Z 850.458,A -85,B 0,C 180,E1 2156.223,E2 2156.223} C_VEL
LIN {X 0,Y 591.925,Z 845.247,A -85,B 0,C 180,E1 2154.67,E2 2154.67} C_VEL
LIN {X 0,Y 591.939,Z 838.432,A -85,B 0,C 180,E1 2153.21,E2 2153.21} C_VEL
LIN {X 0,Y 591.97,Z 829.91,A -85,B 0,C 180,E1 2151.802,E2 2151.802} C_VEL
LIN {X 0,Y 592.006,Z 819.973,A -85,B 0,C 180,E1 2150.52,E2 2150.52} C_VEL
LIN {X 0,Y 592.059,Z 809.127,A -85,B 0,C 180,E1 2149.382,E2 2149.382} C_VEL
LIN {X 0,Y 592.123,Z 796.405,A -85,B 0,C 180,E1 2148.309,E2 2148.309} C_VEL
LIN {X 0,Y 592.176,Z 782.958,A -85,B 0,C 180,E1 2147.403,E2 2147.403} C_VEL
LIN {X 0,Y 592.257,Z 768.304,A -85,B 0,C 180,E1 2146.628,E2 2146.628} C_VEL
LIN {X 0,Y 592.318,Z 752.475,A -85,B 0,C 180,E1 2146.007,E2 2146.007} C_VEL
LIN {X 0,Y 592.364,Z 736.555,A -85,B 0,C 180,E1 2145.571,E2 2145.571} C_VEL
LIN {X 0,Y 592.407,Z 716.508,A -85,B 0,C 180,E1 2145.266,E2 2145.266} C_VEL
LIN {X 0,Y 592.329,Z 588.301,A -85,B 0,C 180,E1 2143.677,E2 2143.677} C_VEL
LIN {X 0,Y 592.518,Z 541.742,A -85,B 0,C 180,E1 2140.533,E2 2140.533} C_VEL
LIN {X 0,Y 592.724,Z 495.931,A -85,B 0,C 180,E1 2137.381,E2 2137.381} C_VEL
LIN {X 0,Y 592.971,Z 451.545,A -85,B 0,C 180,E1 2134.261,E2 2134.261} C_VEL
LIN {X 0,Y 593.244,Z 419.705,A -85,B 0,C 180,E1 2131.951,E2 2131.951} C_VEL
LIN {X 0,Y 595.992,Z 382.776,A -85,B 0,C 180,E1 2128.776,E2 2128.776} C_VEL
LIN {X 0,Y 596.368,Z 365.909,A -85,B 0,C 180,E1 2127.058,E2 2127.058} C_VEL
LIN {X 0,Y 594.248,Z 361.592,A -85,B 0,C 180,E1 2126.221,E2 2126.221} C_VEL
LIN {X 0,Y 592.298,Z 358.295,A -85,B 0,C 180,E1 2125.445,E2 2125.445} C_VEL
LIN {X 0,Y 592.029,Z 356.993,A -85,B 0,C 180,E1 2125.165,E2 2125.165} C_VEL
LIN {X 0,Y 592.036,Z 356.993,A -85,B 0,C 180,E1 2121.907,E2 2121.907} C_VEL
LIN {X 0,Y 592.029,Z 357.022,A -85,B 0,C 180,E1 2120.454,E2 2120.454} C_VEL
LIN {X 0,Y 593.266,Z 360.367,A -85,B 0,C 180,E1 2120.051,E2 2120.051} C_VEL
LIN {X 0,Y 594.441,Z 362.462,A -85,B 0,C 180,E1 2119.786,E2 2119.786} C_VEL
LIN {X 0,Y 594.779,Z 363.774,A -85,B 0,C 180,E1 2119.669,E2 2119.669} C_VEL
LIN {X 0,Y 593.888,Z 392.827,A -85,B 0,C 180,E1 2118.058,E2 2118.058} C_VEL
LIN {X 0,Y 594.031,Z 426.956,A -85,B 0,C 180,E1 2116.296,E2 2116.296} C_VEL
LIN {X 0,Y 595.539,Z 441,A -85,B 0,C 180,E1 2115.504,E2 2115.504} C_VEL
LIN {X 0,Y 597.568,Z 449.53,A -85,B 0,C 180,E1 2114.919,E2 2114.919} C_VEL
LIN {X 0,Y 599.298,Z 454.303,A -85,B 0,C 180,E1 2114.434,E2 2114.434} C_VEL
LIN {X 0,Y 600.997,Z 457.386,A -85,B 0,C 180,E1 2113.916,E2 2113.916} C_VEL
LIN {X 0,Y 602.389,Z 458.782,A -85,B 0,C 180,E1 2113.365,E2 2113.365} C_VEL
LIN {X 0,Y 603.133,Z 458.511,A -85,B 0,C 180,E1 2112.82,E2 2112.82} C_VEL
LIN {X 0,Y 603.112,Z 456.554,A -85,B 0,C 180,E1 2112.306,E2 2112.306} C_VEL
LIN {X 0,Y 602.3,Z 453.007,A -85,B 0,C 180,E1 2111.863,E2 2111.863} C_VEL
LIN {X 0,Y 600.838,Z 447.94,A -85,B 0,C 180,E1 2111.525,E2 2111.525} C_VEL
LIN {X 0,Y 598.921,Z 440.651,A -85,B 0,C 180,E1 2111.292,E2 2111.292} C_VEL
LIN {X 0,Y 597.614,Z 430.41,A -85,B 0,C 180,E1 2111.149,E2 2111.149} C_VEL
LIN {X 0,Y 597.269,Z 420.635,A -85,B 0,C 180,E1 2111.112,E2 2111.112} C_VEL
LIN {X 0,Y 597.172,Z 364.554,A -85,B 0,C 180,E1 2111.101,E2 2111.101} C_VEL
LIN {X 0,Y 596.105,Z 363.004,A -85,B 0,C 180,E1 2110.983,E2 2110.983} C_VEL
LIN {X 0,Y 593.408,Z 360.591,A -85,B 0,C 180,E1 2110.683,E2 2110.683} C_VEL
LIN {X 0,Y 592.106,Z 357.563,A -85,B 0,C 180,E1 2110.536,E2 2110.536} C_VEL
LIN {X 0,Y 592.013,Z 356.993,A -85,B 0,C 180,E1 2110.517,E2 2110.517} C_VEL
LIN {X 0,Y 592.028,Z 357.037,A -85,B 0,C 180,E1 2108.922,E2 2108.922} C_VEL
LIN {X 0,Y 592.987,Z 359.921,A -85,B 0,C 180,E1 2108.677,E2 2108.677} C_VEL
LIN {X 0,Y 594.593,Z 363.341,A -85,B 0,C 180,E1 2108.353,E2 2108.353} C_VEL
LIN {X 0,Y 594.218,Z 415.877,A -85,B 0,C 180,E1 2105.369,E2 2105.369} C_VEL
LIN {X 0,Y 594.072,Z 455.33,A -85,B 0,C 180,E1 2103.218,E2 2103.218} C_VEL
LIN {X 0,Y 594.371,Z 461.426,A -85,B 0,C 180,E1 2103.113,E2 2103.113} C_VEL
LIN {X 0,Y 593.988,Z 677.68,A -85,B 0,C 180,E1 2100.129,E2 2100.129} C_VEL
LIN {X 0,Y 593.808,Z 761.957,A -85,B 0,C 180,E1 2098.96,E2 2098.96} C_VEL
LIN {X 0,Y 593.692,Z 783.553,A -85,B 0,C 180,E1 2098.472,E2 2098.472} C_VEL
LIN {X 0,Y 593.518,Z 805.516,A -85,B 0,C 180,E1 2097.79,E2 2097.79} C_VEL
LIN {X 0,Y 593.357,Z 826.49,A -85,B 0,C 180,E1 2096.949,E2 2096.949} C_VEL
LIN {X 0,Y 593.168,Z 846.736,A -85,B 0,C 180,E1 2095.94,E2 2095.94} C_VEL
LIN {X 0,Y 592.944,Z 867.138,A -85,B 0,C 180,E1 2094.721,E2 2094.721} C_VEL
LIN {X 0,Y 592.765,Z 885.586,A -85,B 0,C 180,E1 2093.423,E2 2093.423} C_VEL
LIN {X 0,Y 592.578,Z 904.101,A -85,B 0,C 180,E1 2091.895,E2 2091.895} C_VEL
LIN {X 0,Y 592.404,Z 921.216,A -85,B 0,C 180,E1 2090.243,E2 2090.243} C_VEL
LIN {X 0,Y 592.247,Z 936.721,A -85,B 0,C 180,E1 2088.506,E2 2088.506} C_VEL
LIN {X 0,Y 592.139,Z 950.745,A -85,B 0,C 180,E1 2086.682,E2 2086.682} C_VEL
LIN {X 0,Y 592.059,Z 963.342,A -85,B 0,C 180,E1 2084.774,E2 2084.774} C_VEL
LIN {X 0,Y 591.993,Z 973.85,A -85,B 0,C 180,E1 2082.882,E2 2082.882} C_VEL
LIN {X 0,Y 591.948,Z 983.478,A -85,B 0,C 180,E1 2080.807,E2 2080.807} C_VEL
LIN {X 0,Y 591.931,Z 990.972,A -85,B 0,C 180,E1 2078.831,E2 2078.831} C_VEL
LIN {X 0,Y 591.919,Z 996.913,A -85,B 0,C 180,E1 2076.791,E2 2076.791} C_VEL
LIN {X 0,Y 591.906,Z 1001.468,A -85,B 0,C 180,E1 2074.651,E2 2074.651} C_VEL
LIN {X 0,Y 591.894,Z 1004.238,A -85,B 0,C 180,E1 2072.614,E2 2072.614} C_VEL
LIN {X 0,Y 591.891,Z 1005.373,A -85,B 0,C 180,E1 2070.581,E2 2070.581} C_VEL
LIN {X 0,Y 591.9,Z 1005.086,A -85,B 0,C 180,E1 2068.548,E2 2068.548} C_VEL
LIN {X 0,Y 591.913,Z 1003.228,A -85,B 0,C 180,E1 2066.514,E2 2066.514} C_VEL
LIN {X 0,Y 591.918,Z 999.609,A -85,B 0,C 180,E1 2064.378,E2 2064.378} C_VEL
LIN {X 0,Y 591.915,Z 994.588,A -85,B 0,C 180,E1 2062.331,E2 2062.331} C_VEL
LIN {X 0,Y 591.919,Z 988.115,A -85,B 0,C 180,E1 2060.374,E2 2060.374} C_VEL
LIN {X 0,Y 591.953,Z 979.607,A -85,B 0,C 180,E1 2058.306,E2 2058.306} C_VEL
LIN {X 0,Y 592.002,Z 970.218,A -85,B 0,C 180,E1 2056.423,E2 2056.423} C_VEL
LIN {X 0,Y 592.068,Z 958.911,A -85,B 0,C 180,E1 2054.525,E2 2054.525} C_VEL
LIN {X 0,Y 592.175,Z 945.57,A -85,B 0,C 180,E1 2052.611,E2 2052.611} C_VEL
LIN {X 0,Y 592.307,Z 931.589,A -85,B 0,C 180,E1 2050.884,E2 2050.884} C_VEL
LIN {X 0,Y 592.463,Z 915.146,A -85,B 0,C 180,E1 2049.14,E2 2049.14} C_VEL
LIN {X 0,Y 592.62,Z 898.081,A -85,B 0,C 180,E1 2047.586,E2 2047.586} C_VEL
LIN {X 0,Y 592.816,Z 879.389,A -85,B 0,C 180,E1 2046.122,E2 2046.122} C_VEL
LIN {X 0,Y 593.038,Z 860.539,A -85,B 0,C 180,E1 2044.858,E2 2044.858} C_VEL
LIN {X 0,Y 593.223,Z 840.44,A -85,B 0,C 180,E1 2043.723,E2 2043.723} C_VEL
LIN {X 0,Y 593.406,Z 820.194,A -85,B 0,C 180,E1 2042.782,E2 2042.782} C_VEL
LIN {X 0,Y 593.59,Z 798.863,A -85,B 0,C 180,E1 2041.983,E2 2041.983} C_VEL
LIN {X 0,Y 593.712,Z 777.606,A -85,B 0,C 180,E1 2041.372,E2 2041.372} C_VEL
LIN {X 0,Y 593.826,Z 756.149,A -85,B 0,C 180,E1 2040.946,E2 2040.946} C_VEL
LIN {X 0,Y 594.255,Z 523.641,A -85,B 0,C 180,E1 2037.755,E2 2037.755} C_VEL
LIN {X 0,Y 594.173,Z 455.966,A -85,B 0,C 180,E1 2036.797,E2 2036.797} C_VEL
LIN {X 0,Y 593.97,Z 453.716,A -85,B 0,C 180,E1 2036.717,E2 2036.717} C_VEL
LIN {X 0,Y 594.344,Z 399.067,A -85,B 0,C 180,E1 2033.689,E2 2033.689} C_VEL
LIN {X 0,Y 594.593,Z 363.353,A -85,B 0,C 180,E1 2031.647,E2 2031.647} C_VEL
LIN {X 0,Y 592.121,Z 357.597,A -85,B 0,C 180,E1 2031.118,E2 2031.118} C_VEL
LIN {X 0,Y 592.023,Z 356.992,A -85,B 0,C 180,E1 2031.037,E2 2031.037} C_VEL
LIN {X 0,Y 592.022,Z 357.061,A -85,B 0,C 180,E1 2029.474,E2 2029.474} C_VEL
LIN {X 0,Y 593.079,Z 360.085,A -85,B 0,C 180,E1 2029.354,E2 2029.354} C_VEL
LIN {X 0,Y 595.61,Z 362.705,A -85,B 0,C 180,E1 2029.072,E2 2029.072} C_VEL
LIN {X 0,Y 596.676,Z 363.662,A -85,B 0,C 180,E1 2028.954,E2 2028.954} C_VEL
LIN {X 0,Y 597.263,Z 364.705,A -85,B 0,C 180,E1 2028.889,E2 2028.889} C_VEL
LIN {X 0,Y 597.45,Z 427.645,A -85,B 0,C 180,E1 2028.868,E2 2028.868} C_VEL
LIN {X 0,Y 598.546,Z 438.582,A -85,B 0,C 180,E1 2028.749,E2 2028.749} C_VEL
LIN {X 0,Y 600.454,Z 446.64,A -85,B 0,C 180,E1 2028.533,E2 2028.533} C_VEL
LIN {X 0,Y 602.038,Z 452.053,A -85,B 0,C 180,E1 2028.218,E2 2028.218} C_VEL
LIN {X 0,Y 603.018,Z 456.012,A -85,B 0,C 180,E1 2027.783,E2 2027.783} C_VEL
LIN {X 0,Y 603.202,Z 458.177,A -85,B 0,C 180,E1 2027.316,E2 2027.316} C_VEL
LIN {X 0,Y 602.796,Z 458.872,A -85,B 0,C 180,E1 2026.872,E2 2026.872} C_VEL
LIN {X 0,Y 601.606,Z 458.137,A -85,B 0,C 180,E1 2026.299,E2 2026.299} C_VEL
LIN {X 0,Y 600,Z 455.752,A -85,B 0,C 180,E1 2025.771,E2 2025.771} C_VEL
LIN {X 0,Y 598.035,Z 451.015,A -85,B 0,C 180,E1 2025.212,E2 2025.212} C_VEL
LIN {X 0,Y 596.111,Z 442.329,A -85,B 0,C 180,E1 2024.516,E2 2024.516} C_VEL
LIN {X 0,Y 595.282,Z 429.054,A -85,B 0,C 180,E1 2023.621,E2 2023.621} C_VEL
LIN {X 0,Y 595.608,Z 384.334,A -85,B 0,C 180,E1 2020.791,E2 2020.791} C_VEL
LIN {X 0,Y 595.778,Z 364.974,A -85,B 0,C 180,E1 2019.498,E2 2019.498} C_VEL
LIN {X 0,Y 593.85,Z 361.149,A -85,B 0,C 180,E1 2019.028,E2 2019.028} C_VEL
LIN {X 0,Y 592.28,Z 358.225,A -85,B 0,C 180,E1 2018.654,E2 2018.654} C_VEL
LIN {X 0,Y 592.029,Z 356.991,A -85,B 0,C 180,E1 2018.524,E2 2018.524} C_VEL
LIN {X 0,Y 591.986,Z 356.994,A -85,B 0,C 180,E1 2015.284,E2 2015.284} C_VEL
LIN {X 0,Y 592.038,Z 356.988,A -85,B 0,C 180,E1 2012.139,E2 2012.139} C_VEL
LIN {X 0,Y 591.998,Z 356.992,A -85,B 0,C 180,E1 2008.884,E2 2008.884} C_VEL
LIN {X 0,Y 592.017,Z 356.989,A -85,B 0,C 180,E1 2005.595,E2 2005.595} C_VEL
LIN {X 0,Y 592.012,Z 356.99,A -85,B 0,C 180,E1 2002.438,E2 2002.438} C_VEL
LIN {X 0,Y 591.995,Z 356.992,A -85,B 0,C 180,E1 1999.229,E2 1999.229} C_VEL
LIN {X 0,Y 592.029,Z 356.99,A -85,B 0,C 180,E1 1996.18,E2 1996.18} C_VEL
LIN {X 0,Y 592.016,Z 356.993,A -85,B 0,C 180,E1 1992.968,E2 1992.968} C_VEL
LIN {X 0,Y 592.035,Z 356.992,A -85,B 0,C 180,E1 1989.821,E2 1989.821} C_VEL
LIN {X 0,Y 592.03,Z 356.993,A -85,B 0,C 180,E1 1986.594,E2 1986.594} C_VEL
LIN {X 0,Y 592.04,Z 356.991,A -85,B 0,C 180,E1 1983.291,E2 1983.291} C_VEL
LIN {X 0,Y 592.025,Z 356.992,A -85,B 0,C 180,E1 1980,E2 1980} C_VEL
LIN {X 0,Y 592.021,Z 356.993,A -85,B 0,C 180,E1 1976.75,E2 1976.75} C_VEL
LIN {X 0,Y 592.029,Z 356.992,A -85,B 0,C 180,E1 1973.503,E2 1973.503} C_VEL
LIN {X 0,Y 592.019,Z 356.993,A -85,B 0,C 180,E1 1970.276,E2 1970.276} C_VEL
LIN {X 0,Y 592.002,Z 356.993,A -85,B 0,C 180,E1 1970.107,E2 1970.107} C_VEL
LIN {X 0,Y 590.981,Z 357.119,A -85,B 0,C 180,E1 1969.362,E2 1969.362} C_VEL
LIN {X 0,Y 584.617,Z 357.917,A -85,B 0,C 180,E1 1967.269,E2 1967.269} C_VEL
LIN {X 0,Y 584.096,Z 357.977,A -85,B 0,C 180,E1 1966.725,E2 1966.725} C_VEL
LIN {X 0,Y 584.057,Z 357.981,A -85,B 0,C 180,E1 1963.47,E2 1963.47} C_VEL
LIN {X 0,Y 584.087,Z 357.977,A -85,B 0,C 180,E1 1960.187,E2 1960.187} C_VEL
LIN {X 0,Y 584.071,Z 357.979,A -85,B 0,C 180,E1 1957.026,E2 1957.026} C_VEL
LIN {X 0,Y 584.065,Z 357.98,A -85,B 0,C 180,E1 1953.77,E2 1953.77} C_VEL
LIN {X 0,Y 584.084,Z 357.979,A -85,B 0,C 180,E1 1950.613,E2 1950.613} C_VEL
LIN {X 0,Y 584.061,Z 357.982,A -85,B 0,C 180,E1 1947.367,E2 1947.367} C_VEL
LIN {X 0,Y 584.094,Z 357.973,A -85,B 0,C 180,E1 1944.232,E2 1944.232} C_VEL
LIN {X 0,Y 584.069,Z 357.982,A -85,B 0,C 180,E1 1940.951,E2 1940.951} C_VEL
LIN {X 0,Y 584.097,Z 357.975,A -85,B 0,C 180,E1 1937.688,E2 1937.688} C_VEL
LIN {X 0,Y 584.075,Z 357.98,A -85,B 0,C 180,E1 1934.439,E2 1934.439} C_VEL
LIN {X 0,Y 584.084,Z 357.981,A -85,B 0,C 180,E1 1931.228,E2 1931.228} C_VEL
LIN {X 0,Y 584.088,Z 357.981,A -85,B 0,C 180,E1 1928.043,E2 1928.043} C_VEL
LIN {X 0,Y 584.083,Z 357.983,A -85,B 0,C 180,E1 1924.872,E2 1924.872} C_VEL
LIN {X 0,Y 584.095,Z 357.982,A -85,B 0,C 180,E1 1921.703,E2 1921.703} C_VEL
LIN {X 0,Y 584.097,Z 358.004,A -85,B 0,C 180,E1 1921.243,E2 1921.243} C_VEL
LIN {X 0,Y 586.196,Z 364.394,A -85,B 0,C 180,E1 1920.663,E2 1920.663} C_VEL
LIN {X 0,Y 585.78,Z 409.674,A -85,B 0,C 180,E1 1917.497,E2 1917.497} C_VEL
LIN {X 0,Y 585.37,Z 455.752,A -85,B 0,C 180,E1 1914.362,E2 1914.362} C_VEL
LIN {X 0,Y 585.317,Z 473.548,A -85,B 0,C 180,E1 1913.191,E2 1913.191} C_VEL
LIN {X 0,Y 585.738,Z 479.624,A -85,B 0,C 180,E1 1913.094,E2 1913.094} C_VEL
LIN {X 0,Y 585.335,Z 682.862,A -85,B 0,C 180,E1 1910.452,E2 1910.452} C_VEL
LIN {X 0,Y 585.224,Z 702.076,A -85,B 0,C 180,E1 1910.012,E2 1910.012} C_VEL
LIN {X 0,Y 585.082,Z 720.252,A -85,B 0,C 180,E1 1909.408,E2 1909.408} C_VEL
LIN {X 0,Y 584.888,Z 737.715,A -85,B 0,C 180,E1 1908.643,E2 1908.643} C_VEL
LIN {X 0,Y 584.747,Z 754.409,A -85,B 0,C 180,E1 1907.72,E2 1907.72} C_VEL
LIN {X 0,Y 584.558,Z 770.895,A -85,B 0,C 180,E1 1906.597,E2 1906.597} C_VEL
LIN {X 0,Y 584.384,Z 786.243,A -85,B 0,C 180,E1 1905.328,E2 1905.328} C_VEL
LIN {X 0,Y 584.238,Z 799.974,A -85,B 0,C 180,E1 1903.963,E2 1903.963} C_VEL
LIN {X 0,Y 584.126,Z 812.623,A -85,B 0,C 180,E1 1902.455,E2 1902.455} C_VEL
LIN {X 0,Y 584.04,Z 823.726,A -85,B 0,C 180,E1 1900.854,E2 1900.854} C_VEL
LIN {X 0,Y 583.976,Z 833.299,A -85,B 0,C 180,E1 1899.162,E2 1899.162} C_VEL
LIN {X 0,Y 583.943,Z 840.905,A -85,B 0,C 180,E1 1897.477,E2 1897.477} C_VEL
LIN {X 0,Y 583.917,Z 847.078,A -85,B 0,C 180,E1 1895.699,E2 1895.699} C_VEL
LIN {X 0,Y 583.919,Z 851.484,A -85,B 0,C 180,E1 1893.927,E2 1893.927} C_VEL
LIN {X 0,Y 583.916,Z 854.349,A -85,B 0,C 180,E1 1892.06,E2 1892.06} C_VEL
LIN {X 0,Y 583.911,Z 855.452,A -85,B 0,C 180,E1 1890.196,E2 1890.196} C_VEL
LIN {X 0,Y 583.913,Z 854.812,A -85,B 0,C 180,E1 1888.332,E2 1888.332} C_VEL
LIN {X 0,Y 583.907,Z 852.419,A -85,B 0,C 180,E1 1886.465,E2 1886.465} C_VEL
LIN {X 0,Y 583.917,Z 848.459,A -85,B 0,C 180,E1 1884.694,E2 1884.694} C_VEL
LIN {X 0,Y 583.932,Z 842.777,A -85,B 0,C 180,E1 1882.918,E2 1882.918} C_VEL
LIN {X 0,Y 583.958,Z 835.676,A -85,B 0,C 180,E1 1881.234,E2 1881.234} C_VEL
LIN {X 0,Y 584.016,Z 826.699,A -85,B 0,C 180,E1 1879.544,E2 1879.544} C_VEL
LIN {X 0,Y 584.092,Z 816.263,A -85,B 0,C 180,E1 1877.945,E2 1877.945} C_VEL
LIN {X 0,Y 584.201,Z 804.385,A -85,B 0,C 180,E1 1876.439,E2 1876.439} C_VEL
LIN {X 0,Y 584.345,Z 791.031,A -85,B 0,C 180,E1 1875.026,E2 1875.026} C_VEL
LIN {X 0,Y 584.506,Z 775.998,A -85,B 0,C 180,E1 1873.707,E2 1873.707} C_VEL
LIN {X 0,Y 584.679,Z 760.601,A -85,B 0,C 180,E1 1872.586,E2 1872.586} C_VEL
LIN {X 0,Y 584.83,Z 743.398,A -85,B 0,C 180,E1 1871.561,E2 1871.561} C_VEL
LIN {X 0,Y 585.027,Z 726.118,A -85,B 0,C 180,E1 1870.74,E2 1870.74} C_VEL
LIN {X 0,Y 585.19,Z 707.273,A -85,B 0,C 180,E1 1870.054,E2 1870.054} C_VEL
LIN {X 0,Y 585.312,Z 688.055,A -85,B 0,C 180,E1 1869.559,E2 1869.559} C_VEL
LIN {X 0,Y 585.385,Z 665.591,A -85,B 0,C 180,E1 1869.211,E2 1869.211} C_VEL
LIN {X 0,Y 585.568,Z 475.143,A -85,B 0,C 180,E1 1866.75,E2 1866.75} C_VEL
LIN {X 0,Y 585.257,Z 472.831,A -85,B 0,C 180,E1 1866.693,E2 1866.693} C_VEL
LIN {X 0,Y 585.615,Z 426.068,A -85,B 0,C 180,E1 1863.537,E2 1863.537} C_VEL
LIN {X 0,Y 586.053,Z 380.75,A -85,B 0,C 180,E1 1860.402,E2 1860.402} C_VEL
LIN {X 0,Y 585.999,Z 363.613,A -85,B 0,C 180,E1 1859.179,E2 1859.179} C_VEL
LIN {X 0,Y 584.062,Z 357.981,A -85,B 0,C 180,E1 1858.639,E2 1858.639} C_VEL
